Fanuc TP program (LS listing): FM113226.ls

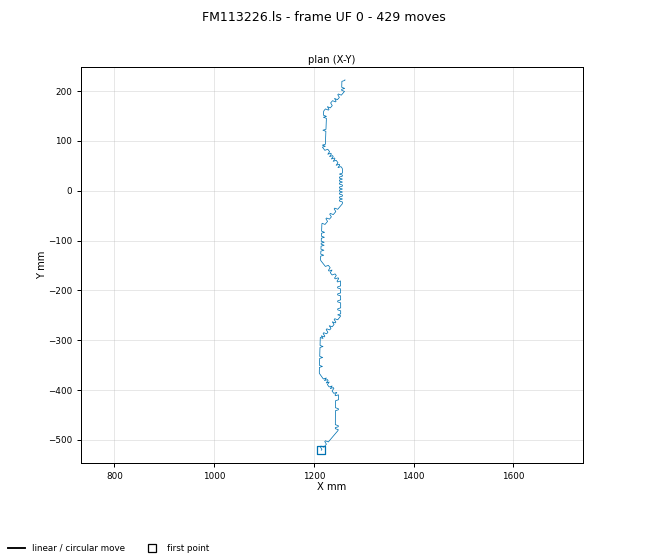
[picture p0: tool path of FM113226.ls in frame UF 0, 429 of 429 moves have a stored position in this frame; points joined in program order, loops and branches not executed]
/PROG  FM113226
/ATTR
OWNER		= MNEDITOR;
COMMENT		= "Auto FANUC move";
PROG_SIZE	= 0;
CREATE		= DATE 26-05-06  TIME 11:32:26;
MODIFIED	= DATE 26-05-06  TIME 11:32:26;
FILE_NAME	= ;
VERSION		= 0;
LINE_COUNT	= 434;
MEMORY_SIZE	= 0;
PROTECT		= READ_WRITE;
TCD:  STACK_SIZE	= 0,
      TASK_PRIORITY	= 50,
      TIME_SLICE	= 0,
      BUSY_LAMP_OFF	= 0,
      ABORT_REQUEST	= 0,
      PAUSE_REQUEST	= 0;
DEFAULT_GROUP	= 1,*,*,*,*;
CONTROL_CODE	= 00000000 00000000;
/MN
   1:  UFRAME_NUM=0 ;
   2:  UTOOL_NUM=1 ;
   3:  R[93]=10 ;
   4:  L P[1] 7mm/sec FINE ;
   5:  L P[2] 7mm/sec CNT50 ;
   6:  L P[3] 7mm/sec CNT50 ;
   7:  L P[4] 7mm/sec CNT50 ;
   8:  L P[5] 7mm/sec CNT50 ;
   9:  L P[6] 7mm/sec CNT50 ;
  10:  L P[7] 7mm/sec CNT50 ;
  11:  L P[8] 7mm/sec CNT50 ;
  12:  L P[9] 7mm/sec CNT50 ;
  13:  L P[10] 7mm/sec CNT50 ;
  14:  L P[11] 7mm/sec CNT50 ;
  15:  L P[12] 7mm/sec CNT50 ;
  16:  L P[13] 7mm/sec CNT50 ;
  17:  L P[14] 7mm/sec CNT50 ;
  18:  L P[15] 7mm/sec CNT50 ;
  19:  L P[16] 7mm/sec CNT50 ;
  20:  L P[17] 7mm/sec CNT50 ;
  21:  L P[18] 7mm/sec CNT50 ;
  22:  L P[19] 7mm/sec CNT50 ;
  23:  L P[20] 7mm/sec CNT50 ;
  24:  L P[21] 7mm/sec CNT50 ;
  25:  L P[22] 7mm/sec CNT50 ;
  26:  L P[23] 7mm/sec CNT50 ;
  27:  L P[24] 7mm/sec CNT50 ;
  28:  L P[25] 7mm/sec CNT50 ;
  29:  L P[26] 7mm/sec CNT50 ;
  30:  L P[27] 7mm/sec CNT50 ;
  31:  L P[28] 7mm/sec CNT50 ;
  32:  L P[29] 7mm/sec CNT50 ;
  33:  L P[30] 7mm/sec CNT50 ;
  34:  L P[31] 7mm/sec CNT50 ;
  35:  L P[32] 7mm/sec CNT50 ;
  36:  L P[33] 7mm/sec CNT50 ;
  37:  L P[34] 7mm/sec CNT50 ;
  38:  L P[35] 7mm/sec CNT50 ;
  39:  L P[36] 7mm/sec CNT50 ;
  40:  L P[37] 7mm/sec CNT50 ;
  41:  L P[38] 7mm/sec CNT50 ;
  42:  L P[39] 7mm/sec CNT50 ;
  43:  L P[40] 7mm/sec CNT50 ;
  44:  L P[41] 7mm/sec CNT50 ;
  45:  L P[42] 7mm/sec CNT50 ;
  46:  L P[43] 7mm/sec CNT50 ;
  47:  L P[44] 7mm/sec CNT50 ;
  48:  L P[45] 7mm/sec CNT50 ;
  49:  L P[46] 7mm/sec CNT50 ;
  50:  L P[47] 7mm/sec CNT50 ;
  51:  L P[48] 7mm/sec CNT50 ;
  52:  L P[49] 7mm/sec CNT50 ;
  53:  L P[50] 7mm/sec CNT50 ;
  54:  L P[51] 7mm/sec CNT50 ;
  55:  L P[52] 7mm/sec CNT50 ;
  56:  L P[53] 7mm/sec CNT50 ;
  57:  L P[54] 7mm/sec CNT50 ;
  58:  L P[55] 7mm/sec CNT50 ;
  59:  L P[56] 7mm/sec CNT50 ;
  60:  L P[57] 7mm/sec CNT50 ;
  61:  L P[58] 7mm/sec CNT50 ;
  62:  L P[59] 7mm/sec CNT50 ;
  63:  L P[60] 7mm/sec CNT50 ;
  64:  L P[61] 7mm/sec CNT50 ;
  65:  L P[62] 7mm/sec CNT50 ;
  66:  L P[63] 7mm/sec CNT50 ;
  67:  L P[64] 7mm/sec CNT50 ;
  68:  L P[65] 7mm/sec CNT50 ;
  69:  L P[66] 7mm/sec CNT50 ;
  70:  L P[67] 7mm/sec CNT50 ;
  71:  L P[68] 7mm/sec CNT50 ;
  72:  L P[69] 7mm/sec CNT50 ;
  73:  L P[70] 7mm/sec CNT50 ;
  74:  L P[71] 7mm/sec CNT50 ;
  75:  L P[72] 7mm/sec CNT50 ;
  76:  L P[73] 7mm/sec CNT50 ;
  77:  L P[74] 7mm/sec CNT50 ;
  78:  L P[75] 7mm/sec CNT50 ;
  79:  L P[76] 7mm/sec CNT50 ;
  80:  L P[77] 7mm/sec CNT50 ;
  81:  L P[78] 7mm/sec CNT50 ;
  82:  L P[79] 7mm/sec CNT50 ;
  83:  L P[80] 7mm/sec CNT50 ;
  84:  L P[81] 7mm/sec CNT50 ;
  85:  L P[82] 7mm/sec CNT50 ;
  86:  L P[83] 7mm/sec CNT50 ;
  87:  L P[84] 7mm/sec CNT50 ;
  88:  L P[85] 7mm/sec CNT50 ;
  89:  L P[86] 7mm/sec CNT50 ;
  90:  L P[87] 7mm/sec CNT50 ;
  91:  L P[88] 7mm/sec CNT50 ;
  92:  L P[89] 7mm/sec CNT50 ;
  93:  L P[90] 7mm/sec CNT50 ;
  94:  L P[91] 7mm/sec CNT50 ;
  95:  L P[92] 7mm/sec CNT50 ;
  96:  L P[93] 7mm/sec CNT50 ;
  97:  L P[94] 7mm/sec CNT50 ;
  98:  L P[95] 7mm/sec CNT50 ;
  99:  L P[96] 7mm/sec CNT50 ;
 100:  L P[97] 7mm/sec CNT50 ;
 101:  L P[98] 7mm/sec CNT50 ;
 102:  L P[99] 7mm/sec CNT50 ;
 103:  L P[100] 7mm/sec CNT50 ;
 104:  L P[101] 7mm/sec CNT50 ;
 105:  L P[102] 7mm/sec CNT50 ;
 106:  L P[103] 7mm/sec CNT50 ;
 107:  L P[104] 7mm/sec CNT50 ;
 108:  L P[105] 7mm/sec CNT50 ;
 109:  L P[106] 7mm/sec CNT50 ;
 110:  L P[107] 7mm/sec CNT50 ;
 111:  L P[108] 7mm/sec CNT50 ;
 112:  L P[109] 7mm/sec CNT50 ;
 113:  L P[110] 7mm/sec CNT50 ;
 114:  L P[111] 7mm/sec CNT50 ;
 115:  L P[112] 7mm/sec CNT50 ;
 116:  L P[113] 7mm/sec CNT50 ;
 117:  L P[114] 7mm/sec CNT50 ;
 118:  L P[115] 7mm/sec CNT50 ;
 119:  L P[116] 7mm/sec CNT50 ;
 120:  L P[117] 7mm/sec CNT50 ;
 121:  L P[118] 7mm/sec CNT50 ;
 122:  L P[119] 7mm/sec CNT50 ;
 123:  L P[120] 7mm/sec CNT50 ;
 124:  L P[121] 7mm/sec CNT50 ;
 125:  L P[122] 7mm/sec CNT50 ;
 126:  L P[123] 7mm/sec CNT50 ;
 127:  L P[124] 7mm/sec CNT50 ;
 128:  L P[125] 7mm/sec CNT50 ;
 129:  L P[126] 7mm/sec CNT50 ;
 130:  L P[127] 7mm/sec CNT50 ;
 131:  L P[128] 7mm/sec CNT50 ;
 132:  L P[129] 7mm/sec CNT50 ;
 133:  L P[130] 7mm/sec CNT50 ;
 134:  L P[131] 7mm/sec CNT50 ;
 135:  L P[132] 7mm/sec CNT50 ;
 136:  L P[133] 7mm/sec CNT50 ;
 137:  L P[134] 7mm/sec CNT50 ;
 138:  L P[135] 7mm/sec CNT50 ;
 139:  L P[136] 7mm/sec CNT50 ;
 140:  L P[137] 7mm/sec CNT50 ;
 141:  L P[138] 7mm/sec CNT50 ;
 142:  L P[139] 7mm/sec CNT50 ;
 143:  L P[140] 7mm/sec CNT50 ;
 144:  L P[141] 7mm/sec CNT50 ;
 145:  L P[142] 7mm/sec CNT50 ;
 146:  L P[143] 7mm/sec CNT50 ;
 147:  L P[144] 7mm/sec CNT50 ;
 148:  L P[145] 7mm/sec CNT50 ;
 149:  L P[146] 7mm/sec CNT50 ;
 150:  L P[147] 7mm/sec CNT50 ;
 151:  L P[148] 7mm/sec CNT50 ;
 152:  L P[149] 7mm/sec CNT50 ;
 153:  L P[150] 7mm/sec CNT50 ;
 154:  L P[151] 7mm/sec CNT50 ;
 155:  L P[152] 7mm/sec CNT50 ;
 156:  L P[153] 7mm/sec CNT50 ;
 157:  L P[154] 7mm/sec CNT50 ;
 158:  L P[155] 7mm/sec CNT50 ;
 159:  L P[156] 7mm/sec CNT50 ;
 160:  L P[157] 7mm/sec CNT50 ;
 161:  L P[158] 7mm/sec CNT50 ;
 162:  L P[159] 7mm/sec CNT50 ;
 163:  L P[160] 7mm/sec CNT50 ;
 164:  L P[161] 7mm/sec CNT50 ;
 165:  L P[162] 7mm/sec CNT50 ;
 166:  L P[163] 7mm/sec CNT50 ;
 167:  L P[164] 7mm/sec CNT50 ;
 168:  L P[165] 7mm/sec CNT50 ;
 169:  L P[166] 7mm/sec CNT50 ;
 170:  L P[167] 7mm/sec CNT50 ;
 171:  L P[168] 7mm/sec CNT50 ;
 172:  L P[169] 7mm/sec CNT50 ;
 173:  L P[170] 7mm/sec CNT50 ;
 174:  L P[171] 7mm/sec CNT50 ;
 175:  L P[172] 7mm/sec CNT50 ;
 176:  L P[173] 7mm/sec CNT50 ;
 177:  L P[174] 7mm/sec CNT50 ;
 178:  L P[175] 7mm/sec CNT50 ;
 179:  L P[176] 7mm/sec CNT50 ;
 180:  L P[177] 7mm/sec CNT50 ;
 181:  L P[178] 7mm/sec CNT50 ;
 182:  L P[179] 7mm/sec CNT50 ;
 183:  L P[180] 7mm/sec CNT50 ;
 184:  L P[181] 7mm/sec CNT50 ;
 185:  L P[182] 7mm/sec CNT50 ;
 186:  L P[183] 7mm/sec CNT50 ;
 187:  L P[184] 7mm/sec CNT50 ;
 188:  L P[185] 7mm/sec CNT50 ;
 189:  L P[186] 7mm/sec CNT50 ;
 190:  L P[187] 7mm/sec CNT50 ;
 191:  L P[188] 7mm/sec CNT50 ;
 192:  L P[189] 7mm/sec CNT50 ;
 193:  L P[190] 7mm/sec CNT50 ;
 194:  L P[191] 7mm/sec CNT50 ;
 195:  L P[192] 7mm/sec CNT50 ;
 196:  L P[193] 7mm/sec CNT50 ;
 197:  L P[194] 7mm/sec CNT50 ;
 198:  L P[195] 7mm/sec CNT50 ;
 199:  L P[196] 7mm/sec CNT50 ;
 200:  L P[197] 7mm/sec CNT50 ;
 201:  L P[198] 7mm/sec CNT50 ;
 202:  L P[199] 7mm/sec CNT50 ;
 203:  L P[200] 7mm/sec CNT50 ;
 204:  L P[201] 7mm/sec CNT50 ;
 205:  L P[202] 7mm/sec CNT50 ;
 206:  L P[203] 7mm/sec CNT50 ;
 207:  L P[204] 7mm/sec CNT50 ;
 208:  L P[205] 7mm/sec CNT50 ;
 209:  L P[206] 7mm/sec CNT50 ;
 210:  L P[207] 7mm/sec CNT50 ;
 211:  L P[208] 7mm/sec CNT50 ;
 212:  L P[209] 7mm/sec CNT50 ;
 213:  L P[210] 7mm/sec CNT50 ;
 214:  L P[211] 7mm/sec CNT50 ;
 215:  L P[212] 7mm/sec CNT50 ;
 216:  L P[213] 7mm/sec CNT50 ;
 217:  L P[214] 7mm/sec CNT50 ;
 218:  L P[215] 7mm/sec CNT50 ;
 219:  L P[216] 7mm/sec CNT50 ;
 220:  L P[217] 7mm/sec CNT50 ;
 221:  L P[218] 7mm/sec CNT50 ;
 222:  L P[219] 7mm/sec CNT50 ;
 223:  L P[220] 7mm/sec CNT50 ;
 224:  L P[221] 7mm/sec CNT50 ;
 225:  L P[222] 7mm/sec CNT50 ;
 226:  L P[223] 7mm/sec CNT50 ;
 227:  L P[224] 7mm/sec CNT50 ;
 228:  L P[225] 7mm/sec CNT50 ;
 229:  L P[226] 7mm/sec CNT50 ;
 230:  L P[227] 7mm/sec CNT50 ;
 231:  L P[228] 7mm/sec CNT50 ;
 232:  L P[229] 7mm/sec CNT50 ;
 233:  L P[230] 7mm/sec CNT50 ;
 234:  L P[231] 7mm/sec CNT50 ;
 235:  L P[232] 7mm/sec CNT50 ;
 236:  L P[233] 7mm/sec CNT50 ;
 237:  L P[234] 7mm/sec CNT50 ;
 238:  L P[235] 7mm/sec CNT50 ;
 239:  L P[236] 7mm/sec CNT50 ;
 240:  L P[237] 7mm/sec CNT50 ;
 241:  L P[238] 7mm/sec CNT50 ;
 242:  L P[239] 7mm/sec CNT50 ;
 243:  L P[240] 7mm/sec CNT50 ;
 244:  L P[241] 7mm/sec CNT50 ;
 245:  L P[242] 7mm/sec CNT50 ;
 246:  L P[243] 7mm/sec CNT50 ;
 247:  L P[244] 7mm/sec CNT50 ;
 248:  L P[245] 7mm/sec CNT50 ;
 249:  L P[246] 7mm/sec CNT50 ;
 250:  L P[247] 7mm/sec CNT50 ;
 251:  L P[248] 7mm/sec CNT50 ;
 252:  L P[249] 7mm/sec CNT50 ;
 253:  L P[250] 7mm/sec CNT50 ;
 254:  L P[251] 7mm/sec CNT50 ;
 255:  L P[252] 7mm/sec CNT50 ;
 256:  L P[253] 7mm/sec CNT50 ;
 257:  L P[254] 7mm/sec CNT50 ;
 258:  L P[255] 7mm/sec CNT50 ;
 259:  L P[256] 7mm/sec CNT50 ;
 260:  L P[257] 7mm/sec CNT50 ;
 261:  L P[258] 7mm/sec CNT50 ;
 262:  L P[259] 7mm/sec CNT50 ;
 263:  L P[260] 7mm/sec CNT50 ;
 264:  L P[261] 7mm/sec CNT50 ;
 265:  L P[262] 7mm/sec CNT50 ;
 266:  L P[263] 7mm/sec CNT50 ;
 267:  L P[264] 7mm/sec CNT50 ;
 268:  L P[265] 7mm/sec CNT50 ;
 269:  L P[266] 7mm/sec CNT50 ;
 270:  L P[267] 7mm/sec CNT50 ;
 271:  L P[268] 7mm/sec CNT50 ;
 272:  L P[269] 7mm/sec CNT50 ;
 273:  L P[270] 7mm/sec CNT50 ;
 274:  L P[271] 7mm/sec CNT50 ;
 275:  L P[272] 7mm/sec CNT50 ;
 276:  L P[273] 7mm/sec CNT50 ;
 277:  L P[274] 7mm/sec CNT50 ;
 278:  L P[275] 7mm/sec CNT50 ;
 279:  L P[276] 7mm/sec CNT50 ;
 280:  L P[277] 7mm/sec CNT50 ;
 281:  L P[278] 7mm/sec CNT50 ;
 282:  L P[279] 7mm/sec CNT50 ;
 283:  L P[280] 7mm/sec CNT50 ;
 284:  L P[281] 7mm/sec CNT50 ;
 285:  L P[282] 7mm/sec CNT50 ;
 286:  L P[283] 7mm/sec CNT50 ;
 287:  L P[284] 7mm/sec CNT50 ;
 288:  L P[285] 7mm/sec CNT50 ;
 289:  L P[286] 7mm/sec CNT50 ;
 290:  L P[287] 7mm/sec CNT50 ;
 291:  L P[288] 7mm/sec CNT50 ;
 292:  L P[289] 7mm/sec CNT50 ;
 293:  L P[290] 7mm/sec CNT50 ;
 294:  L P[291] 7mm/sec CNT50 ;
 295:  L P[292] 7mm/sec CNT50 ;
 296:  L P[293] 7mm/sec CNT50 ;
 297:  L P[294] 7mm/sec CNT50 ;
 298:  L P[295] 7mm/sec CNT50 ;
 299:  L P[296] 7mm/sec CNT50 ;
 300:  L P[297] 7mm/sec CNT50 ;
 301:  L P[298] 7mm/sec CNT50 ;
 302:  L P[299] 7mm/sec CNT50 ;
 303:  L P[300] 7mm/sec CNT50 ;
 304:  L P[301] 7mm/sec CNT50 ;
 305:  L P[302] 7mm/sec CNT50 ;
 306:  L P[303] 7mm/sec CNT50 ;
 307:  L P[304] 7mm/sec CNT50 ;
 308:  L P[305] 7mm/sec CNT50 ;
 309:  L P[306] 7mm/sec CNT50 ;
 310:  L P[307] 7mm/sec CNT50 ;
 311:  L P[308] 7mm/sec CNT50 ;
 312:  L P[309] 7mm/sec CNT50 ;
 313:  L P[310] 7mm/sec CNT50 ;
 314:  L P[311] 7mm/sec CNT50 ;
 315:  L P[312] 7mm/sec CNT50 ;
 316:  L P[313] 7mm/sec CNT50 ;
 317:  L P[314] 7mm/sec CNT50 ;
 318:  L P[315] 7mm/sec CNT50 ;
 319:  L P[316] 7mm/sec CNT50 ;
 320:  L P[317] 7mm/sec CNT50 ;
 321:  L P[318] 7mm/sec CNT50 ;
 322:  L P[319] 7mm/sec CNT50 ;
 323:  L P[320] 7mm/sec CNT50 ;
 324:  L P[321] 7mm/sec CNT50 ;
 325:  L P[322] 7mm/sec CNT50 ;
 326:  L P[323] 7mm/sec CNT50 ;
 327:  L P[324] 7mm/sec CNT50 ;
 328:  L P[325] 7mm/sec CNT50 ;
 329:  L P[326] 7mm/sec CNT50 ;
 330:  L P[327] 7mm/sec CNT50 ;
 331:  L P[328] 7mm/sec CNT50 ;
 332:  L P[329] 7mm/sec CNT50 ;
 333:  L P[330] 7mm/sec CNT50 ;
 334:  L P[331] 7mm/sec CNT50 ;
 335:  L P[332] 7mm/sec CNT50 ;
 336:  L P[333] 7mm/sec CNT50 ;
 337:  L P[334] 7mm/sec CNT50 ;
 338:  L P[335] 7mm/sec CNT50 ;
 339:  L P[336] 7mm/sec CNT50 ;
 340:  L P[337] 7mm/sec CNT50 ;
 341:  L P[338] 7mm/sec CNT50 ;
 342:  L P[339] 7mm/sec CNT50 ;
 343:  L P[340] 7mm/sec CNT50 ;
 344:  L P[341] 7mm/sec CNT50 ;
 345:  L P[342] 7mm/sec CNT50 ;
 346:  L P[343] 7mm/sec CNT50 ;
 347:  L P[344] 7mm/sec CNT50 ;
 348:  L P[345] 7mm/sec CNT50 ;
 349:  L P[346] 7mm/sec CNT50 ;
 350:  L P[347] 7mm/sec CNT50 ;
 351:  L P[348] 7mm/sec CNT50 ;
 352:  L P[349] 7mm/sec CNT50 ;
 353:  L P[350] 7mm/sec CNT50 ;
 354:  L P[351] 7mm/sec CNT50 ;
 355:  L P[352] 7mm/sec CNT50 ;
 356:  L P[353] 7mm/sec CNT50 ;
 357:  L P[354] 7mm/sec CNT50 ;
 358:  L P[355] 7mm/sec CNT50 ;
 359:  L P[356] 7mm/sec CNT50 ;
 360:  L P[357] 7mm/sec CNT50 ;
 361:  L P[358] 7mm/sec CNT50 ;
 362:  L P[359] 7mm/sec CNT50 ;
 363:  L P[360] 7mm/sec CNT50 ;
 364:  L P[361] 7mm/sec CNT50 ;
 365:  L P[362] 7mm/sec CNT50 ;
 366:  L P[363] 7mm/sec CNT50 ;
 367:  L P[364] 7mm/sec CNT50 ;
 368:  L P[365] 7mm/sec CNT50 ;
 369:  L P[366] 7mm/sec CNT50 ;
 370:  L P[367] 7mm/sec CNT50 ;
 371:  L P[368] 7mm/sec CNT50 ;
 372:  L P[369] 7mm/sec CNT50 ;
 373:  L P[370] 7mm/sec CNT50 ;
 374:  L P[371] 7mm/sec CNT50 ;
 375:  L P[372] 7mm/sec CNT50 ;
 376:  L P[373] 7mm/sec CNT50 ;
 377:  L P[374] 7mm/sec CNT50 ;
 378:  L P[375] 7mm/sec CNT50 ;
 379:  L P[376] 7mm/sec CNT50 ;
 380:  L P[377] 7mm/sec CNT50 ;
 381:  L P[378] 7mm/sec CNT50 ;
 382:  L P[379] 7mm/sec CNT50 ;
 383:  L P[380] 7mm/sec CNT50 ;
 384:  L P[381] 7mm/sec CNT50 ;
 385:  L P[382] 7mm/sec CNT50 ;
 386:  L P[383] 7mm/sec CNT50 ;
 387:  L P[384] 7mm/sec CNT50 ;
 388:  L P[385] 7mm/sec CNT50 ;
 389:  L P[386] 7mm/sec CNT50 ;
 390:  L P[387] 7mm/sec CNT50 ;
 391:  L P[388] 7mm/sec CNT50 ;
 392:  L P[389] 7mm/sec CNT50 ;
 393:  L P[390] 7mm/sec CNT50 ;
 394:  L P[391] 7mm/sec CNT50 ;
 395:  L P[392] 7mm/sec CNT50 ;
 396:  L P[393] 7mm/sec CNT50 ;
 397:  L P[394] 7mm/sec CNT50 ;
 398:  L P[395] 7mm/sec CNT50 ;
 399:  L P[396] 7mm/sec CNT50 ;
 400:  L P[397] 7mm/sec CNT50 ;
 401:  L P[398] 7mm/sec CNT50 ;
 402:  L P[399] 7mm/sec CNT50 ;
 403:  L P[400] 7mm/sec CNT50 ;
 404:  L P[401] 7mm/sec CNT50 ;
 405:  L P[402] 7mm/sec CNT50 ;
 406:  L P[403] 7mm/sec CNT50 ;
 407:  L P[404] 7mm/sec CNT50 ;
 408:  L P[405] 7mm/sec CNT50 ;
 409:  L P[406] 7mm/sec CNT50 ;
 410:  L P[407] 7mm/sec CNT50 ;
 411:  L P[408] 7mm/sec CNT50 ;
 412:  L P[409] 7mm/sec CNT50 ;
 413:  L P[410] 7mm/sec CNT50 ;
 414:  L P[411] 7mm/sec CNT50 ;
 415:  L P[412] 7mm/sec CNT50 ;
 416:  L P[413] 7mm/sec CNT50 ;
 417:  L P[414] 7mm/sec CNT50 ;
 418:  L P[415] 7mm/sec CNT50 ;
 419:  L P[416] 7mm/sec CNT50 ;
 420:  L P[417] 7mm/sec CNT50 ;
 421:  L P[418] 7mm/sec CNT50 ;
 422:  L P[419] 7mm/sec CNT50 ;
 423:  L P[420] 7mm/sec CNT50 ;
 424:  L P[421] 7mm/sec CNT50 ;
 425:  L P[422] 7mm/sec CNT50 ;
 426:  L P[423] 7mm/sec CNT50 ;
 427:  L P[424] 7mm/sec CNT50 ;
 428:  L P[425] 7mm/sec CNT50 ;
 429:  L P[426] 7mm/sec CNT50 ;
 430:  L P[427] 7mm/sec CNT50 ;
 431:  L P[428] 7mm/sec CNT50 ;
 432:  L P[429] 7mm/sec FINE ;
 433:  R[93]=1 ;
 434:  END ;
/POS
P[1]{
   GP1:
	UF : 0, UT : 1,		CONFIG : 'N U T, 0, 0, 0',
	X = 1214.854  mm,	Y = -520.674  mm,	Z = -244.012  mm,
	W = 0.000 deg,	P = 30.000 deg,	R = 139.708 deg
};
P[2]{
   GP1:
	UF : 0, UT : 1,		CONFIG : 'N U T, 0, 0, 0',
	X = 1216.138  mm,	Y = -519.161  mm,	Z = -244.261  mm,
	W = 0.000 deg,	P = 30.000 deg,	R = 139.708 deg
};
P[3]{
   GP1:
	UF : 0, UT : 1,		CONFIG : 'N U T, 0, 0, 0',
	X = 1212.844  mm,	Y = -513.767  mm,	Z = -244.510  mm,
	W = 0.000 deg,	P = 30.000 deg,	R = 139.708 deg
};
P[4]{
   GP1:
	UF : 0, UT : 1,		CONFIG : 'N U T, 0, 0, 0',
	X = 1214.128  mm,	Y = -512.253  mm,	Z = -244.760  mm,
	W = 0.000 deg,	P = 30.000 deg,	R = 139.708 deg
};
P[5]{
   GP1:
	UF : 0, UT : 1,		CONFIG : 'N U T, 0, 0, 0',
	X = 1219.987  mm,	Y = -514.620  mm,	Z = -245.009  mm,
	W = 0.000 deg,	P = 30.000 deg,	R = 139.708 deg
};
P[6]{
   GP1:
	UF : 0, UT : 1,		CONFIG : 'N U T, 0, 0, 0',
	X = 1221.271  mm,	Y = -513.106  mm,	Z = -245.258  mm,
	W = 0.000 deg,	P = 30.000 deg,	R = 139.708 deg
};
P[7]{
   GP1:
	UF : 0, UT : 1,		CONFIG : 'N U T, 0, 0, 0',
	X = 1222.554  mm,	Y = -511.593  mm,	Z = -245.507  mm,
	W = 0.000 deg,	P = 30.000 deg,	R = 139.708 deg
};
P[8]{
   GP1:
	UF : 0, UT : 1,		CONFIG : 'N U T, 0, 0, 0',
	X = 1223.837  mm,	Y = -510.079  mm,	Z = -245.756  mm,
	W = 0.000 deg,	P = 30.000 deg,	R = 139.708 deg
};
P[9]{
   GP1:
	UF : 0, UT : 1,		CONFIG : 'N U T, 0, 0, 0',
	X = 1225.121  mm,	Y = -508.565  mm,	Z = -246.005  mm,
	W = 0.000 deg,	P = 30.000 deg,	R = 139.708 deg
};
P[10]{
   GP1:
	UF : 0, UT : 1,		CONFIG : 'N U T, 0, 0, 0',
	X = 1221.827  mm,	Y = -503.171  mm,	Z = -246.254  mm,
	W = 0.000 deg,	P = 30.000 deg,	R = 139.708 deg
};
P[11]{
   GP1:
	UF : 0, UT : 1,		CONFIG : 'N U T, 0, 0, 0',
	X = 1223.111  mm,	Y = -501.658  mm,	Z = -246.503  mm,
	W = 0.000 deg,	P = 30.000 deg,	R = 139.708 deg
};
P[12]{
   GP1:
	UF : 0, UT : 1,		CONFIG : 'N U T, 0, 0, 0',
	X = 1228.970  mm,	Y = -504.024  mm,	Z = -246.752  mm,
	W = 0.000 deg,	P = 30.000 deg,	R = 139.708 deg
};
P[13]{
   GP1:
	UF : 0, UT : 1,		CONFIG : 'N U T, 0, 0, 0',
	X = 1230.254  mm,	Y = -502.511  mm,	Z = -247.001  mm,
	W = 0.000 deg,	P = 30.000 deg,	R = 139.708 deg
};
P[14]{
   GP1:
	UF : 0, UT : 1,		CONFIG : 'N U T, 0, 0, 0',
	X = 1231.537  mm,	Y = -500.997  mm,	Z = -247.250  mm,
	W = 0.000 deg,	P = 30.000 deg,	R = 139.708 deg
};
P[15]{
   GP1:
	UF : 0, UT : 1,		CONFIG : 'N U T, 0, 0, 0',
	X = 1232.820  mm,	Y = -499.483  mm,	Z = -247.499  mm,
	W = 0.000 deg,	P = 30.000 deg,	R = 139.708 deg
};
P[16]{
   GP1:
	UF : 0, UT : 1,		CONFIG : 'N U T, 0, 0, 0',
	X = 1234.104  mm,	Y = -497.970  mm,	Z = -247.748  mm,
	W = 0.000 deg,	P = 30.000 deg,	R = 139.708 deg
};
P[17]{
   GP1:
	UF : 0, UT : 1,		CONFIG : 'N U T, 0, 0, 0',
	X = 1235.387  mm,	Y = -496.456  mm,	Z = -247.997  mm,
	W = 0.000 deg,	P = 30.000 deg,	R = 139.708 deg
};
P[18]{
   GP1:
	UF : 0, UT : 1,		CONFIG : 'N U T, 0, 0, 0',
	X = 1236.670  mm,	Y = -494.942  mm,	Z = -248.246  mm,
	W = 0.000 deg,	P = 30.000 deg,	R = 139.708 deg
};
P[19]{
   GP1:
	UF : 0, UT : 1,		CONFIG : 'N U T, 0, 0, 0',
	X = 1237.954  mm,	Y = -493.429  mm,	Z = -248.495  mm,
	W = 0.000 deg,	P = 30.000 deg,	R = 139.708 deg
};
P[20]{
   GP1:
	UF : 0, UT : 1,		CONFIG : 'N U T, 0, 0, 0',
	X = 1239.237  mm,	Y = -491.915  mm,	Z = -248.744  mm,
	W = 0.000 deg,	P = 30.000 deg,	R = 139.708 deg
};
P[21]{
   GP1:
	UF : 0, UT : 1,		CONFIG : 'N U T, 0, 0, 0',
	X = 1240.520  mm,	Y = -490.401  mm,	Z = -248.993  mm,
	W = 0.000 deg,	P = 30.000 deg,	R = 139.708 deg
};
P[22]{
   GP1:
	UF : 0, UT : 1,		CONFIG : 'N U T, 0, 0, 0',
	X = 1241.803  mm,	Y = -488.888  mm,	Z = -249.242  mm,
	W = 0.000 deg,	P = 30.000 deg,	R = 139.708 deg
};
P[23]{
   GP1:
	UF : 0, UT : 1,		CONFIG : 'N U T, 0, 0, 0',
	X = 1243.087  mm,	Y = -487.374  mm,	Z = -249.492  mm,
	W = 0.000 deg,	P = 30.000 deg,	R = 147.699 deg
};
P[24]{
   GP1:
	UF : 0, UT : 1,		CONFIG : 'N U T, 0, 0, 0',
	X = 1244.370  mm,	Y = -485.861  mm,	Z = -249.741  mm,
	W = 0.000 deg,	P = 30.000 deg,	R = 155.690 deg
};
P[25]{
   GP1:
	UF : 0, UT : 1,		CONFIG : 'N U T, 0, 0, 0',
	X = 1245.653  mm,	Y = -484.347  mm,	Z = -249.990  mm,
	W = 0.000 deg,	P = 30.000 deg,	R = 163.681 deg
};
P[26]{
   GP1:
	UF : 0, UT : 1,		CONFIG : 'N U T, 0, 0, 0',
	X = 1246.937  mm,	Y = -482.833  mm,	Z = -250.239  mm,
	W = 0.000 deg,	P = 30.000 deg,	R = 171.672 deg
};
P[27]{
   GP1:
	UF : 0, UT : 1,		CONFIG : 'N U T, 0, 0, 0',
	X = 1248.220  mm,	Y = -481.320  mm,	Z = -250.488  mm,
	W = 0.000 deg,	P = 30.000 deg,	R = 179.663 deg
};
P[28]{
   GP1:
	UF : 0, UT : 1,		CONFIG : 'N U T, 0, 0, 0',
	X = 1248.981  mm,	Y = -479.414  mm,	Z = -250.498  mm,
	W = 0.000 deg,	P = 30.000 deg,	R = 179.663 deg
};
P[29]{
   GP1:
	UF : 0, UT : 1,		CONFIG : 'N U T, 0, 0, 0',
	X = 1242.994  mm,	Y = -477.381  mm,	Z = -250.475  mm,
	W = 0.000 deg,	P = 30.000 deg,	R = 179.663 deg
};
P[30]{
   GP1:
	UF : 0, UT : 1,		CONFIG : 'N U T, 0, 0, 0',
	X = 1243.005  mm,	Y = -475.381  mm,	Z = -250.452  mm,
	W = 0.000 deg,	P = 30.000 deg,	R = 179.663 deg
};
P[31]{
   GP1:
	UF : 0, UT : 1,		CONFIG : 'N U T, 0, 0, 0',
	X = 1249.017  mm,	Y = -473.417  mm,	Z = -250.429  mm,
	W = 0.000 deg,	P = 30.000 deg,	R = 179.663 deg
};
P[32]{
   GP1:
	UF : 0, UT : 1,		CONFIG : 'N U T, 0, 0, 0',
	X = 1249.029  mm,	Y = -471.417  mm,	Z = -250.405  mm,
	W = 0.000 deg,	P = 30.000 deg,	R = 179.663 deg
};
P[33]{
   GP1:
	UF : 0, UT : 1,		CONFIG : 'N U T, 0, 0, 0',
	X = 1243.041  mm,	Y = -469.382  mm,	Z = -250.382  mm,
	W = 0.000 deg,	P = 30.000 deg,	R = 179.663 deg
};
P[34]{
   GP1:
	UF : 0, UT : 1,		CONFIG : 'N U T, 0, 0, 0',
	X = 1243.052  mm,	Y = -467.382  mm,	Z = -250.359  mm,
	W = 0.000 deg,	P = 30.000 deg,	R = 179.663 deg
};
P[35]{
   GP1:
	UF : 0, UT : 1,		CONFIG : 'N U T, 0, 0, 0',
	X = 1243.064  mm,	Y = -465.382  mm,	Z = -250.336  mm,
	W = 0.000 deg,	P = 30.000 deg,	R = 179.663 deg
};
P[36]{
   GP1:
	UF : 0, UT : 1,		CONFIG : 'N U T, 0, 0, 0',
	X = 1243.076  mm,	Y = -463.382  mm,	Z = -250.312  mm,
	W = 0.000 deg,	P = 30.000 deg,	R = 179.663 deg
};
P[37]{
   GP1:
	UF : 0, UT : 1,		CONFIG : 'N U T, 0, 0, 0',
	X = 1243.088  mm,	Y = -461.383  mm,	Z = -250.289  mm,
	W = 0.000 deg,	P = 30.000 deg,	R = 179.663 deg
};
P[38]{
   GP1:
	UF : 0, UT : 1,		CONFIG : 'N U T, 0, 0, 0',
	X = 1243.100  mm,	Y = -459.383  mm,	Z = -250.266  mm,
	W = 0.000 deg,	P = 30.000 deg,	R = 179.663 deg
};
P[39]{
   GP1:
	UF : 0, UT : 1,		CONFIG : 'N U T, 0, 0, 0',
	X = 1243.111  mm,	Y = -457.383  mm,	Z = -250.243  mm,
	W = 0.000 deg,	P = 30.000 deg,	R = 179.663 deg
};
P[40]{
   GP1:
	UF : 0, UT : 1,		CONFIG : 'N U T, 0, 0, 0',
	X = 1243.123  mm,	Y = -455.383  mm,	Z = -250.219  mm,
	W = 0.000 deg,	P = 30.000 deg,	R = 179.663 deg
};
P[41]{
   GP1:
	UF : 0, UT : 1,		CONFIG : 'N U T, 0, 0, 0',
	X = 1243.135  mm,	Y = -453.383  mm,	Z = -250.196  mm,
	W = 0.000 deg,	P = 30.000 deg,	R = 179.663 deg
};
P[42]{
   GP1:
	UF : 0, UT : 1,		CONFIG : 'N U T, 0, 0, 0',
	X = 1243.147  mm,	Y = -451.383  mm,	Z = -250.173  mm,
	W = 0.000 deg,	P = 30.000 deg,	R = 179.663 deg
};
P[43]{
   GP1:
	UF : 0, UT : 1,		CONFIG : 'N U T, 0, 0, 0',
	X = 1243.158  mm,	Y = -449.384  mm,	Z = -250.149  mm,
	W = 0.000 deg,	P = 30.000 deg,	R = 179.663 deg
};
P[44]{
   GP1:
	UF : 0, UT : 1,		CONFIG : 'N U T, 0, 0, 0',
	X = 1243.170  mm,	Y = -447.384  mm,	Z = -250.126  mm,
	W = 0.000 deg,	P = 30.000 deg,	R = 179.663 deg
};
P[45]{
   GP1:
	UF : 0, UT : 1,		CONFIG : 'N U T, 0, 0, 0',
	X = 1243.182  mm,	Y = -445.384  mm,	Z = -250.103  mm,
	W = 0.000 deg,	P = 30.000 deg,	R = 179.663 deg
};
P[46]{
   GP1:
	UF : 0, UT : 1,		CONFIG : 'N U T, 0, 0, 0',
	X = 1243.194  mm,	Y = -443.384  mm,	Z = -250.080  mm,
	W = 0.000 deg,	P = 30.000 deg,	R = 179.663 deg
};
P[47]{
   GP1:
	UF : 0, UT : 1,		CONFIG : 'N U T, 0, 0, 0',
	X = 1243.205  mm,	Y = -441.384  mm,	Z = -250.056  mm,
	W = 0.000 deg,	P = 30.000 deg,	R = 179.663 deg
};
P[48]{
   GP1:
	UF : 0, UT : 1,		CONFIG : 'N U T, 0, 0, 0',
	X = 1249.217  mm,	Y = -439.420  mm,	Z = -250.033  mm,
	W = 0.000 deg,	P = 30.000 deg,	R = 179.663 deg
};
P[49]{
   GP1:
	UF : 0, UT : 1,		CONFIG : 'N U T, 0, 0, 0',
	X = 1249.229  mm,	Y = -437.420  mm,	Z = -250.010  mm,
	W = 0.000 deg,	P = 30.000 deg,	R = 179.663 deg
};
P[50]{
   GP1:
	UF : 0, UT : 1,		CONFIG : 'N U T, 0, 0, 0',
	X = 1243.241  mm,	Y = -435.385  mm,	Z = -249.987  mm,
	W = 0.000 deg,	P = 30.000 deg,	R = 179.663 deg
};
P[51]{
   GP1:
	UF : 0, UT : 1,		CONFIG : 'N U T, 0, 0, 0',
	X = 1243.253  mm,	Y = -433.385  mm,	Z = -249.963  mm,
	W = 0.000 deg,	P = 30.000 deg,	R = 179.663 deg
};
P[52]{
   GP1:
	UF : 0, UT : 1,		CONFIG : 'N U T, 0, 0, 0',
	X = 1243.264  mm,	Y = -431.385  mm,	Z = -249.940  mm,
	W = 0.000 deg,	P = 30.000 deg,	R = 179.663 deg
};
P[53]{
   GP1:
	UF : 0, UT : 1,		CONFIG : 'N U T, 0, 0, 0',
	X = 1243.276  mm,	Y = -429.385  mm,	Z = -249.917  mm,
	W = 0.000 deg,	P = 30.000 deg,	R = 179.663 deg
};
P[54]{
   GP1:
	UF : 0, UT : 1,		CONFIG : 'N U T, 0, 0, 0',
	X = 1243.288  mm,	Y = -427.385  mm,	Z = -249.894  mm,
	W = 0.000 deg,	P = 30.000 deg,	R = 179.663 deg
};
P[55]{
   GP1:
	UF : 0, UT : 1,		CONFIG : 'N U T, 0, 0, 0',
	X = 1243.300  mm,	Y = -425.386  mm,	Z = -249.870  mm,
	W = 0.000 deg,	P = 30.000 deg,	R = 179.663 deg
};
P[56]{
   GP1:
	UF : 0, UT : 1,		CONFIG : 'N U T, 0, 0, 0',
	X = 1243.311  mm,	Y = -423.386  mm,	Z = -249.847  mm,
	W = 0.000 deg,	P = 30.000 deg,	R = 179.663 deg
};
P[57]{
   GP1:
	UF : 0, UT : 1,		CONFIG : 'N U T, 0, 0, 0',
	X = 1243.323  mm,	Y = -421.386  mm,	Z = -249.824  mm,
	W = 0.000 deg,	P = 30.000 deg,	R = 179.663 deg
};
P[58]{
   GP1:
	UF : 0, UT : 1,		CONFIG : 'N U T, 0, 0, 0',
	X = 1249.335  mm,	Y = -419.421  mm,	Z = -249.800  mm,
	W = 0.000 deg,	P = 30.000 deg,	R = -173.342 deg
};
P[59]{
   GP1:
	UF : 0, UT : 1,		CONFIG : 'N U T, 0, 0, 0',
	X = 1249.347  mm,	Y = -417.422  mm,	Z = -249.777  mm,
	W = 0.000 deg,	P = 30.000 deg,	R = -166.059 deg
};
P[60]{
   GP1:
	UF : 0, UT : 1,		CONFIG : 'N U T, 0, 0, 0',
	X = 1249.358  mm,	Y = -415.422  mm,	Z = -249.754  mm,
	W = 0.000 deg,	P = 30.000 deg,	R = -158.776 deg
};
P[61]{
   GP1:
	UF : 0, UT : 1,		CONFIG : 'N U T, 0, 0, 0',
	X = 1249.370  mm,	Y = -413.422  mm,	Z = -249.731  mm,
	W = 0.000 deg,	P = 30.000 deg,	R = -151.493 deg
};
P[62]{
   GP1:
	UF : 0, UT : 1,		CONFIG : 'N U T, 0, 0, 0',
	X = 1249.382  mm,	Y = -411.422  mm,	Z = -249.707  mm,
	W = 0.000 deg,	P = 30.000 deg,	R = -144.211 deg
};
P[63]{
   GP1:
	UF : 0, UT : 1,		CONFIG : 'N U T, 0, 0, 0',
	X = 1249.288  mm,	Y = -409.480  mm,	Z = -249.694  mm,
	W = 0.000 deg,	P = 30.000 deg,	R = -143.923 deg
};
P[64]{
   GP1:
	UF : 0, UT : 1,		CONFIG : 'N U T, 0, 0, 0',
	X = 1243.470  mm,	Y = -411.339  mm,	Z = -249.584  mm,
	W = 0.000 deg,	P = 30.000 deg,	R = -143.923 deg
};
P[65]{
   GP1:
	UF : 0, UT : 1,		CONFIG : 'N U T, 0, 0, 0',
	X = 1242.302  mm,	Y = -409.737  mm,	Z = -249.324  mm,
	W = 0.000 deg,	P = 30.000 deg,	R = -143.923 deg
};
P[66]{
   GP1:
	UF : 0, UT : 1,		CONFIG : 'N U T, 0, 0, 0',
	X = 1245.984  mm,	Y = -404.601  mm,	Z = -249.064  mm,
	W = 0.000 deg,	P = 30.000 deg,	R = -143.923 deg
};
P[67]{
   GP1:
	UF : 0, UT : 1,		CONFIG : 'N U T, 0, 0, 0',
	X = 1239.967  mm,	Y = -406.531  mm,	Z = -248.804  mm,
	W = 0.000 deg,	P = 30.000 deg,	R = -143.923 deg
};
P[68]{
   GP1:
	UF : 0, UT : 1,		CONFIG : 'N U T, 0, 0, 0',
	X = 1238.799  mm,	Y = -404.928  mm,	Z = -248.545  mm,
	W = 0.000 deg,	P = 30.000 deg,	R = -143.923 deg
};
P[69]{
   GP1:
	UF : 0, UT : 1,		CONFIG : 'N U T, 0, 0, 0',
	X = 1237.631  mm,	Y = -403.325  mm,	Z = -248.285  mm,
	W = 0.000 deg,	P = 30.000 deg,	R = -143.923 deg
};
P[70]{
   GP1:
	UF : 0, UT : 1,		CONFIG : 'N U T, 0, 0, 0',
	X = 1236.464  mm,	Y = -401.723  mm,	Z = -248.025  mm,
	W = 0.000 deg,	P = 30.000 deg,	R = -143.923 deg
};
P[71]{
   GP1:
	UF : 0, UT : 1,		CONFIG : 'N U T, 0, 0, 0',
	X = 1240.145  mm,	Y = -396.587  mm,	Z = -247.765  mm,
	W = 0.000 deg,	P = 30.000 deg,	R = -143.923 deg
};
P[72]{
   GP1:
	UF : 0, UT : 1,		CONFIG : 'N U T, 0, 0, 0',
	X = 1238.977  mm,	Y = -394.984  mm,	Z = -247.505  mm,
	W = 0.000 deg,	P = 30.000 deg,	R = -143.923 deg
};
P[73]{
   GP1:
	UF : 0, UT : 1,		CONFIG : 'N U T, 0, 0, 0',
	X = 1232.960  mm,	Y = -396.914  mm,	Z = -247.245  mm,
	W = 0.000 deg,	P = 30.000 deg,	R = -143.923 deg
};
P[74]{
   GP1:
	UF : 0, UT : 1,		CONFIG : 'N U T, 0, 0, 0',
	X = 1236.642  mm,	Y = -391.778  mm,	Z = -246.985  mm,
	W = 0.000 deg,	P = 30.000 deg,	R = -143.923 deg
};
P[75]{
   GP1:
	UF : 0, UT : 1,		CONFIG : 'N U T, 0, 0, 0',
	X = 1230.625  mm,	Y = -393.709  mm,	Z = -246.726  mm,
	W = 0.000 deg,	P = 30.000 deg,	R = -143.923 deg
};
P[76]{
   GP1:
	UF : 0, UT : 1,		CONFIG : 'N U T, 0, 0, 0',
	X = 1229.457  mm,	Y = -392.106  mm,	Z = -246.466  mm,
	W = 0.000 deg,	P = 30.000 deg,	R = -143.923 deg
};
P[77]{
   GP1:
	UF : 0, UT : 1,		CONFIG : 'N U T, 0, 0, 0',
	X = 1228.289  mm,	Y = -390.503  mm,	Z = -246.206  mm,
	W = 0.000 deg,	P = 30.000 deg,	R = -143.923 deg
};
P[78]{
   GP1:
	UF : 0, UT : 1,		CONFIG : 'N U T, 0, 0, 0',
	X = 1227.121  mm,	Y = -388.901  mm,	Z = -245.946  mm,
	W = 0.000 deg,	P = 30.000 deg,	R = -143.923 deg
};
P[79]{
   GP1:
	UF : 0, UT : 1,		CONFIG : 'N U T, 0, 0, 0',
	X = 1230.803  mm,	Y = -383.765  mm,	Z = -245.686  mm,
	W = 0.000 deg,	P = 30.000 deg,	R = -143.923 deg
};
P[80]{
   GP1:
	UF : 0, UT : 1,		CONFIG : 'N U T, 0, 0, 0',
	X = 1224.786  mm,	Y = -385.695  mm,	Z = -245.426  mm,
	W = 0.000 deg,	P = 30.000 deg,	R = -143.923 deg
};
P[81]{
   GP1:
	UF : 0, UT : 1,		CONFIG : 'N U T, 0, 0, 0',
	X = 1228.468  mm,	Y = -380.559  mm,	Z = -245.166  mm,
	W = 0.000 deg,	P = 30.000 deg,	R = -143.923 deg
};
P[82]{
   GP1:
	UF : 0, UT : 1,		CONFIG : 'N U T, 0, 0, 0',
	X = 1227.300  mm,	Y = -378.956  mm,	Z = -244.907  mm,
	W = 0.000 deg,	P = 30.000 deg,	R = -143.923 deg
};
P[83]{
   GP1:
	UF : 0, UT : 1,		CONFIG : 'N U T, 0, 0, 0',
	X = 1221.283  mm,	Y = -380.887  mm,	Z = -244.647  mm,
	W = 0.000 deg,	P = 30.000 deg,	R = -143.923 deg
};
P[84]{
   GP1:
	UF : 0, UT : 1,		CONFIG : 'N U T, 0, 0, 0',
	X = 1224.964  mm,	Y = -375.751  mm,	Z = -244.387  mm,
	W = 0.000 deg,	P = 30.000 deg,	R = -143.923 deg
};
P[85]{
   GP1:
	UF : 0, UT : 1,		CONFIG : 'N U T, 0, 0, 0',
	X = 1218.947  mm,	Y = -377.681  mm,	Z = -244.127  mm,
	W = 0.000 deg,	P = 30.000 deg,	R = -143.923 deg
};
P[86]{
   GP1:
	UF : 0, UT : 1,		CONFIG : 'N U T, 0, 0, 0',
	X = 1217.779  mm,	Y = -376.079  mm,	Z = -243.867  mm,
	W = 0.000 deg,	P = 30.000 deg,	R = -143.923 deg
};
P[87]{
   GP1:
	UF : 0, UT : 1,		CONFIG : 'N U T, 0, 0, 0',
	X = 1216.612  mm,	Y = -374.476  mm,	Z = -243.607  mm,
	W = 0.000 deg,	P = 30.000 deg,	R = -154.648 deg
};
P[88]{
   GP1:
	UF : 0, UT : 1,		CONFIG : 'N U T, 0, 0, 0',
	X = 1215.444  mm,	Y = -372.873  mm,	Z = -243.347  mm,
	W = 0.000 deg,	P = 30.000 deg,	R = -162.185 deg
};
P[89]{
   GP1:
	UF : 0, UT : 1,		CONFIG : 'N U T, 0, 0, 0',
	X = 1214.276  mm,	Y = -371.270  mm,	Z = -243.088  mm,
	W = 0.000 deg,	P = 30.000 deg,	R = -169.721 deg
};
P[90]{
   GP1:
	UF : 0, UT : 1,		CONFIG : 'N U T, 0, 0, 0',
	X = 1213.108  mm,	Y = -369.668  mm,	Z = -242.828  mm,
	W = 0.000 deg,	P = 30.000 deg,	R = -177.258 deg
};
P[91]{
   GP1:
	UF : 0, UT : 1,		CONFIG : 'N U T, 0, 0, 0',
	X = 1211.941  mm,	Y = -368.065  mm,	Z = -242.568  mm,
	W = 0.000 deg,	P = 30.000 deg,	R = 178.394 deg
};
P[92]{
   GP1:
	UF : 0, UT : 1,		CONFIG : 'N U T, 0, 0, 0',
	X = 1210.932  mm,	Y = -366.371  mm,	Z = -242.446  mm,
	W = 0.000 deg,	P = 30.000 deg,	R = 178.394 deg
};
P[93]{
   GP1:
	UF : 0, UT : 1,		CONFIG : 'N U T, 0, 0, 0',
	X = 1210.847  mm,	Y = -364.401  mm,	Z = -242.440  mm,
	W = 0.000 deg,	P = 30.000 deg,	R = 178.394 deg
};
P[94]{
   GP1:
	UF : 0, UT : 1,		CONFIG : 'N U T, 0, 0, 0',
	X = 1210.903  mm,	Y = -362.402  mm,	Z = -242.428  mm,
	W = 0.000 deg,	P = 30.000 deg,	R = 178.394 deg
};
P[95]{
   GP1:
	UF : 0, UT : 1,		CONFIG : 'N U T, 0, 0, 0',
	X = 1210.959  mm,	Y = -360.403  mm,	Z = -242.416  mm,
	W = 0.000 deg,	P = 30.000 deg,	R = 178.394 deg
};
P[96]{
   GP1:
	UF : 0, UT : 1,		CONFIG : 'N U T, 0, 0, 0',
	X = 1211.016  mm,	Y = -358.404  mm,	Z = -242.404  mm,
	W = 0.000 deg,	P = 30.000 deg,	R = 178.394 deg
};
P[97]{
   GP1:
	UF : 0, UT : 1,		CONFIG : 'N U T, 0, 0, 0',
	X = 1211.072  mm,	Y = -356.405  mm,	Z = -242.393  mm,
	W = 0.000 deg,	P = 30.000 deg,	R = 178.394 deg
};
P[98]{
   GP1:
	UF : 0, UT : 1,		CONFIG : 'N U T, 0, 0, 0',
	X = 1211.128  mm,	Y = -354.405  mm,	Z = -242.381  mm,
	W = 0.000 deg,	P = 30.000 deg,	R = 178.394 deg
};
P[99]{
   GP1:
	UF : 0, UT : 1,		CONFIG : 'N U T, 0, 0, 0',
	X = 1217.181  mm,	Y = -352.574  mm,	Z = -242.369  mm,
	W = 0.000 deg,	P = 30.000 deg,	R = 178.394 deg
};
P[100]{
   GP1:
	UF : 0, UT : 1,		CONFIG : 'N U T, 0, 0, 0',
	X = 1211.240  mm,	Y = -350.407  mm,	Z = -242.358  mm,
	W = 0.000 deg,	P = 30.000 deg,	R = 178.394 deg
};
P[101]{
   GP1:
	UF : 0, UT : 1,		CONFIG : 'N U T, 0, 0, 0',
	X = 1211.296  mm,	Y = -348.408  mm,	Z = -242.346  mm,
	W = 0.000 deg,	P = 30.000 deg,	R = 178.394 deg
};
P[102]{
   GP1:
	UF : 0, UT : 1,		CONFIG : 'N U T, 0, 0, 0',
	X = 1211.352  mm,	Y = -346.409  mm,	Z = -242.334  mm,
	W = 0.000 deg,	P = 30.000 deg,	R = 178.394 deg
};
P[103]{
   GP1:
	UF : 0, UT : 1,		CONFIG : 'N U T, 0, 0, 0',
	X = 1211.408  mm,	Y = -344.410  mm,	Z = -242.323  mm,
	W = 0.000 deg,	P = 30.000 deg,	R = 178.394 deg
};
P[104]{
   GP1:
	UF : 0, UT : 1,		CONFIG : 'N U T, 0, 0, 0',
	X = 1211.464  mm,	Y = -342.410  mm,	Z = -242.311  mm,
	W = 0.000 deg,	P = 30.000 deg,	R = 178.394 deg
};
P[105]{
   GP1:
	UF : 0, UT : 1,		CONFIG : 'N U T, 0, 0, 0',
	X = 1211.520  mm,	Y = -340.411  mm,	Z = -242.299  mm,
	W = 0.000 deg,	P = 30.000 deg,	R = 178.394 deg
};
P[106]{
   GP1:
	UF : 0, UT : 1,		CONFIG : 'N U T, 0, 0, 0',
	X = 1211.576  mm,	Y = -338.412  mm,	Z = -242.288  mm,
	W = 0.000 deg,	P = 30.000 deg,	R = 178.394 deg
};
P[107]{
   GP1:
	UF : 0, UT : 1,		CONFIG : 'N U T, 0, 0, 0',
	X = 1211.632  mm,	Y = -336.413  mm,	Z = -242.276  mm,
	W = 0.000 deg,	P = 30.000 deg,	R = 178.394 deg
};
P[108]{
   GP1:
	UF : 0, UT : 1,		CONFIG : 'N U T, 0, 0, 0',
	X = 1217.686  mm,	Y = -334.582  mm,	Z = -242.264  mm,
	W = 0.000 deg,	P = 30.000 deg,	R = 178.394 deg
};
P[109]{
   GP1:
	UF : 0, UT : 1,		CONFIG : 'N U T, 0, 0, 0',
	X = 1211.744  mm,	Y = -332.414  mm,	Z = -242.252  mm,
	W = 0.000 deg,	P = 30.000 deg,	R = 178.394 deg
};
P[110]{
   GP1:
	UF : 0, UT : 1,		CONFIG : 'N U T, 0, 0, 0',
	X = 1211.800  mm,	Y = -330.415  mm,	Z = -242.241  mm,
	W = 0.000 deg,	P = 30.000 deg,	R = 178.394 deg
};
P[111]{
   GP1:
	UF : 0, UT : 1,		CONFIG : 'N U T, 0, 0, 0',
	X = 1211.856  mm,	Y = -328.416  mm,	Z = -242.229  mm,
	W = 0.000 deg,	P = 30.000 deg,	R = 178.394 deg
};
P[112]{
   GP1:
	UF : 0, UT : 1,		CONFIG : 'N U T, 0, 0, 0',
	X = 1211.912  mm,	Y = -326.417  mm,	Z = -242.217  mm,
	W = 0.000 deg,	P = 30.000 deg,	R = 178.394 deg
};
P[113]{
   GP1:
	UF : 0, UT : 1,		CONFIG : 'N U T, 0, 0, 0',
	X = 1211.968  mm,	Y = -324.418  mm,	Z = -242.206  mm,
	W = 0.000 deg,	P = 30.000 deg,	R = 178.394 deg
};
P[114]{
   GP1:
	UF : 0, UT : 1,		CONFIG : 'N U T, 0, 0, 0',
	X = 1212.024  mm,	Y = -322.419  mm,	Z = -242.194  mm,
	W = 0.000 deg,	P = 30.000 deg,	R = 178.394 deg
};
P[115]{
   GP1:
	UF : 0, UT : 1,		CONFIG : 'N U T, 0, 0, 0',
	X = 1212.080  mm,	Y = -320.419  mm,	Z = -242.182  mm,
	W = 0.000 deg,	P = 30.000 deg,	R = 178.394 deg
};
P[116]{
   GP1:
	UF : 0, UT : 1,		CONFIG : 'N U T, 0, 0, 0',
	X = 1212.136  mm,	Y = -318.420  mm,	Z = -242.171  mm,
	W = 0.000 deg,	P = 30.000 deg,	R = 178.394 deg
};
P[117]{
   GP1:
	UF : 0, UT : 1,		CONFIG : 'N U T, 0, 0, 0',
	X = 1212.192  mm,	Y = -316.421  mm,	Z = -242.159  mm,
	W = 0.000 deg,	P = 30.000 deg,	R = 178.394 deg
};
P[118]{
   GP1:
	UF : 0, UT : 1,		CONFIG : 'N U T, 0, 0, 0',
	X = 1212.249  mm,	Y = -314.422  mm,	Z = -242.147  mm,
	W = 0.000 deg,	P = 30.000 deg,	R = 178.394 deg
};
P[119]{
   GP1:
	UF : 0, UT : 1,		CONFIG : 'N U T, 0, 0, 0',
	X = 1218.302  mm,	Y = -312.591  mm,	Z = -242.135  mm,
	W = 0.000 deg,	P = 30.000 deg,	R = 178.394 deg
};
P[120]{
   GP1:
	UF : 0, UT : 1,		CONFIG : 'N U T, 0, 0, 0',
	X = 1212.361  mm,	Y = -310.423  mm,	Z = -242.124  mm,
	W = 0.000 deg,	P = 30.000 deg,	R = 178.394 deg
};
P[121]{
   GP1:
	UF : 0, UT : 1,		CONFIG : 'N U T, 0, 0, 0',
	X = 1212.417  mm,	Y = -308.424  mm,	Z = -242.112  mm,
	W = 0.000 deg,	P = 30.000 deg,	R = 178.394 deg
};
P[122]{
   GP1:
	UF : 0, UT : 1,		CONFIG : 'N U T, 0, 0, 0',
	X = 1212.473  mm,	Y = -306.425  mm,	Z = -242.100  mm,
	W = 0.000 deg,	P = 30.000 deg,	R = 178.394 deg
};
P[123]{
   GP1:
	UF : 0, UT : 1,		CONFIG : 'N U T, 0, 0, 0',
	X = 1212.529  mm,	Y = -304.426  mm,	Z = -242.089  mm,
	W = 0.000 deg,	P = 30.000 deg,	R = 174.516 deg
};
P[124]{
   GP1:
	UF : 0, UT : 1,		CONFIG : 'N U T, 0, 0, 0',
	X = 1212.585  mm,	Y = -302.427  mm,	Z = -242.077  mm,
	W = 0.000 deg,	P = 30.000 deg,	R = 167.199 deg
};
P[125]{
   GP1:
	UF : 0, UT : 1,		CONFIG : 'N U T, 0, 0, 0',
	X = 1212.641  mm,	Y = -300.428  mm,	Z = -242.065  mm,
	W = 0.000 deg,	P = 30.000 deg,	R = 159.881 deg
};
P[126]{
   GP1:
	UF : 0, UT : 1,		CONFIG : 'N U T, 0, 0, 0',
	X = 1212.697  mm,	Y = -298.428  mm,	Z = -242.054  mm,
	W = 0.000 deg,	P = 30.000 deg,	R = 152.564 deg
};
P[127]{
   GP1:
	UF : 0, UT : 1,		CONFIG : 'N U T, 0, 0, 0',
	X = 1212.753  mm,	Y = -296.429  mm,	Z = -242.042  mm,
	W = 0.000 deg,	P = 30.000 deg,	R = 145.247 deg
};
P[128]{
   GP1:
	UF : 0, UT : 1,		CONFIG : 'N U T, 0, 0, 0',
	X = 1212.819  mm,	Y = -294.456  mm,	Z = -242.032  mm,
	W = 0.000 deg,	P = 30.000 deg,	R = 141.808 deg
};
P[129]{
   GP1:
	UF : 0, UT : 1,		CONFIG : 'N U T, 0, 0, 0',
	X = 1218.332  mm,	Y = -296.431  mm,	Z = -242.065  mm,
	W = 0.000 deg,	P = 30.000 deg,	R = 141.808 deg
};
P[130]{
   GP1:
	UF : 0, UT : 1,		CONFIG : 'N U T, 0, 0, 0',
	X = 1214.845  mm,	Y = -291.160  mm,	Z = -242.297  mm,
	W = 0.000 deg,	P = 30.000 deg,	R = 141.808 deg
};
P[131]{
   GP1:
	UF : 0, UT : 1,		CONFIG : 'N U T, 0, 0, 0',
	X = 1220.789  mm,	Y = -293.309  mm,	Z = -242.528  mm,
	W = 0.000 deg,	P = 30.000 deg,	R = 141.808 deg
};
P[132]{
   GP1:
	UF : 0, UT : 1,		CONFIG : 'N U T, 0, 0, 0',
	X = 1222.017  mm,	Y = -291.747  mm,	Z = -242.760  mm,
	W = 0.000 deg,	P = 30.000 deg,	R = 141.808 deg
};
P[133]{
   GP1:
	UF : 0, UT : 1,		CONFIG : 'N U T, 0, 0, 0',
	X = 1218.530  mm,	Y = -286.476  mm,	Z = -242.992  mm,
	W = 0.000 deg,	P = 30.000 deg,	R = 141.808 deg
};
P[134]{
   GP1:
	UF : 0, UT : 1,		CONFIG : 'N U T, 0, 0, 0',
	X = 1219.758  mm,	Y = -284.915  mm,	Z = -243.224  mm,
	W = 0.000 deg,	P = 30.000 deg,	R = 141.808 deg
};
P[135]{
   GP1:
	UF : 0, UT : 1,		CONFIG : 'N U T, 0, 0, 0',
	X = 1225.702  mm,	Y = -287.063  mm,	Z = -243.455  mm,
	W = 0.000 deg,	P = 30.000 deg,	R = 141.808 deg
};
P[136]{
   GP1:
	UF : 0, UT : 1,		CONFIG : 'N U T, 0, 0, 0',
	X = 1226.930  mm,	Y = -285.502  mm,	Z = -243.687  mm,
	W = 0.000 deg,	P = 30.000 deg,	R = 141.808 deg
};
P[137]{
   GP1:
	UF : 0, UT : 1,		CONFIG : 'N U T, 0, 0, 0',
	X = 1228.158  mm,	Y = -283.941  mm,	Z = -243.919  mm,
	W = 0.000 deg,	P = 30.000 deg,	R = 141.808 deg
};
P[138]{
   GP1:
	UF : 0, UT : 1,		CONFIG : 'N U T, 0, 0, 0',
	X = 1224.671  mm,	Y = -278.670  mm,	Z = -244.151  mm,
	W = 0.000 deg,	P = 30.000 deg,	R = 141.808 deg
};
P[139]{
   GP1:
	UF : 0, UT : 1,		CONFIG : 'N U T, 0, 0, 0',
	X = 1225.899  mm,	Y = -277.108  mm,	Z = -244.383  mm,
	W = 0.000 deg,	P = 30.000 deg,	R = 141.808 deg
};
P[140]{
   GP1:
	UF : 0, UT : 1,		CONFIG : 'N U T, 0, 0, 0',
	X = 1231.843  mm,	Y = -279.257  mm,	Z = -244.614  mm,
	W = 0.000 deg,	P = 30.000 deg,	R = 141.808 deg
};
P[141]{
   GP1:
	UF : 0, UT : 1,		CONFIG : 'N U T, 0, 0, 0',
	X = 1233.071  mm,	Y = -277.696  mm,	Z = -244.846  mm,
	W = 0.000 deg,	P = 30.000 deg,	R = 141.808 deg
};
P[142]{
   GP1:
	UF : 0, UT : 1,		CONFIG : 'N U T, 0, 0, 0',
	X = 1234.300  mm,	Y = -276.134  mm,	Z = -245.078  mm,
	W = 0.000 deg,	P = 30.000 deg,	R = 141.808 deg
};
P[143]{
   GP1:
	UF : 0, UT : 1,		CONFIG : 'N U T, 0, 0, 0',
	X = 1230.812  mm,	Y = -270.863  mm,	Z = -245.310  mm,
	W = 0.000 deg,	P = 30.000 deg,	R = 141.808 deg
};
P[144]{
   GP1:
	UF : 0, UT : 1,		CONFIG : 'N U T, 0, 0, 0',
	X = 1236.756  mm,	Y = -273.012  mm,	Z = -245.541  mm,
	W = 0.000 deg,	P = 30.000 deg,	R = 141.808 deg
};
P[145]{
   GP1:
	UF : 0, UT : 1,		CONFIG : 'N U T, 0, 0, 0',
	X = 1237.984  mm,	Y = -271.450  mm,	Z = -245.773  mm,
	W = 0.000 deg,	P = 30.000 deg,	R = 141.808 deg
};
P[146]{
   GP1:
	UF : 0, UT : 1,		CONFIG : 'N U T, 0, 0, 0',
	X = 1239.213  mm,	Y = -269.889  mm,	Z = -246.005  mm,
	W = 0.000 deg,	P = 30.000 deg,	R = 141.808 deg
};
P[147]{
   GP1:
	UF : 0, UT : 1,		CONFIG : 'N U T, 0, 0, 0',
	X = 1240.441  mm,	Y = -268.328  mm,	Z = -246.237  mm,
	W = 0.000 deg,	P = 30.000 deg,	R = 141.808 deg
};
P[148]{
   GP1:
	UF : 0, UT : 1,		CONFIG : 'N U T, 0, 0, 0',
	X = 1236.954  mm,	Y = -263.057  mm,	Z = -246.468  mm,
	W = 0.000 deg,	P = 30.000 deg,	R = 141.808 deg
};
P[149]{
   GP1:
	UF : 0, UT : 1,		CONFIG : 'N U T, 0, 0, 0',
	X = 1242.898  mm,	Y = -265.205  mm,	Z = -246.700  mm,
	W = 0.000 deg,	P = 30.000 deg,	R = 141.808 deg
};
P[150]{
   GP1:
	UF : 0, UT : 1,		CONFIG : 'N U T, 0, 0, 0',
	X = 1244.126  mm,	Y = -263.644  mm,	Z = -246.932  mm,
	W = 0.000 deg,	P = 30.000 deg,	R = 141.808 deg
};
P[151]{
   GP1:
	UF : 0, UT : 1,		CONFIG : 'N U T, 0, 0, 0',
	X = 1240.638  mm,	Y = -258.373  mm,	Z = -247.164  mm,
	W = 0.000 deg,	P = 30.000 deg,	R = 141.808 deg
};
P[152]{
   GP1:
	UF : 0, UT : 1,		CONFIG : 'N U T, 0, 0, 0',
	X = 1241.867  mm,	Y = -256.812  mm,	Z = -247.396  mm,
	W = 0.000 deg,	P = 30.000 deg,	R = 141.808 deg
};
P[153]{
   GP1:
	UF : 0, UT : 1,		CONFIG : 'N U T, 0, 0, 0',
	X = 1247.811  mm,	Y = -258.960  mm,	Z = -247.627  mm,
	W = 0.000 deg,	P = 30.000 deg,	R = 150.585 deg
};
P[154]{
   GP1:
	UF : 0, UT : 1,		CONFIG : 'N U T, 0, 0, 0',
	X = 1249.039  mm,	Y = -257.399  mm,	Z = -247.859  mm,
	W = 0.000 deg,	P = 30.000 deg,	R = 158.269 deg
};
P[155]{
   GP1:
	UF : 0, UT : 1,		CONFIG : 'N U T, 0, 0, 0',
	X = 1250.267  mm,	Y = -255.838  mm,	Z = -248.091  mm,
	W = 0.000 deg,	P = 30.000 deg,	R = 165.953 deg
};
P[156]{
   GP1:
	UF : 0, UT : 1,		CONFIG : 'N U T, 0, 0, 0',
	X = 1251.495  mm,	Y = -254.276  mm,	Z = -248.323  mm,
	W = 0.000 deg,	P = 30.000 deg,	R = 173.637 deg
};
P[157]{
   GP1:
	UF : 0, UT : 1,		CONFIG : 'N U T, 0, 0, 0',
	X = 1252.724  mm,	Y = -252.715  mm,	Z = -248.554  mm,
	W = 0.000 deg,	P = 30.000 deg,	R = -179.771 deg
};
P[158]{
   GP1:
	UF : 0, UT : 1,		CONFIG : 'N U T, 0, 0, 0',
	X = 1253.729  mm,	Y = -250.992  mm,	Z = -248.639  mm,
	W = 0.000 deg,	P = 30.000 deg,	R = -179.771 deg
};
P[159]{
   GP1:
	UF : 0, UT : 1,		CONFIG : 'N U T, 0, 0, 0',
	X = 1247.807  mm,	Y = -249.032  mm,	Z = -248.614  mm,
	W = 0.000 deg,	P = 30.000 deg,	R = -179.771 deg
};
P[160]{
   GP1:
	UF : 0, UT : 1,		CONFIG : 'N U T, 0, 0, 0',
	X = 1253.799  mm,	Y = -247.008  mm,	Z = -248.574  mm,
	W = 0.000 deg,	P = 30.000 deg,	R = -179.771 deg
};
P[161]{
   GP1:
	UF : 0, UT : 1,		CONFIG : 'N U T, 0, 0, 0',
	X = 1253.791  mm,	Y = -245.008  mm,	Z = -248.535  mm,
	W = 0.000 deg,	P = 30.000 deg,	R = -179.771 deg
};
P[162]{
   GP1:
	UF : 0, UT : 1,		CONFIG : 'N U T, 0, 0, 0',
	X = 1253.783  mm,	Y = -243.009  mm,	Z = -248.496  mm,
	W = 0.000 deg,	P = 30.000 deg,	R = -179.771 deg
};
P[163]{
   GP1:
	UF : 0, UT : 1,		CONFIG : 'N U T, 0, 0, 0',
	X = 1253.775  mm,	Y = -241.009  mm,	Z = -248.457  mm,
	W = 0.000 deg,	P = 30.000 deg,	R = -179.771 deg
};
P[164]{
   GP1:
	UF : 0, UT : 1,		CONFIG : 'N U T, 0, 0, 0',
	X = 1247.767  mm,	Y = -239.034  mm,	Z = -248.418  mm,
	W = 0.000 deg,	P = 30.000 deg,	R = -179.771 deg
};
P[165]{
   GP1:
	UF : 0, UT : 1,		CONFIG : 'N U T, 0, 0, 0',
	X = 1247.759  mm,	Y = -237.034  mm,	Z = -248.378  mm,
	W = 0.000 deg,	P = 30.000 deg,	R = -179.771 deg
};
P[166]{
   GP1:
	UF : 0, UT : 1,		CONFIG : 'N U T, 0, 0, 0',
	X = 1253.751  mm,	Y = -235.010  mm,	Z = -248.339  mm,
	W = 0.000 deg,	P = 30.000 deg,	R = -179.771 deg
};
P[167]{
   GP1:
	UF : 0, UT : 1,		CONFIG : 'N U T, 0, 0, 0',
	X = 1253.743  mm,	Y = -233.011  mm,	Z = -248.300  mm,
	W = 0.000 deg,	P = 30.000 deg,	R = -179.771 deg
};
P[168]{
   GP1:
	UF : 0, UT : 1,		CONFIG : 'N U T, 0, 0, 0',
	X = 1253.735  mm,	Y = -231.011  mm,	Z = -248.261  mm,
	W = 0.000 deg,	P = 30.000 deg,	R = -179.771 deg
};
P[169]{
   GP1:
	UF : 0, UT : 1,		CONFIG : 'N U T, 0, 0, 0',
	X = 1253.727  mm,	Y = -229.012  mm,	Z = -248.222  mm,
	W = 0.000 deg,	P = 30.000 deg,	R = -179.771 deg
};
P[170]{
   GP1:
	UF : 0, UT : 1,		CONFIG : 'N U T, 0, 0, 0',
	X = 1253.719  mm,	Y = -227.012  mm,	Z = -248.182  mm,
	W = 0.000 deg,	P = 30.000 deg,	R = -179.771 deg
};
P[171]{
   GP1:
	UF : 0, UT : 1,		CONFIG : 'N U T, 0, 0, 0',
	X = 1253.711  mm,	Y = -225.012  mm,	Z = -248.143  mm,
	W = 0.000 deg,	P = 30.000 deg,	R = -179.771 deg
};
P[172]{
   GP1:
	UF : 0, UT : 1,		CONFIG : 'N U T, 0, 0, 0',
	X = 1247.703  mm,	Y = -223.037  mm,	Z = -248.104  mm,
	W = 0.000 deg,	P = 30.000 deg,	R = -179.771 deg
};
P[173]{
   GP1:
	UF : 0, UT : 1,		CONFIG : 'N U T, 0, 0, 0',
	X = 1247.695  mm,	Y = -221.037  mm,	Z = -248.065  mm,
	W = 0.000 deg,	P = 30.000 deg,	R = -179.771 deg
};
P[174]{
   GP1:
	UF : 0, UT : 1,		CONFIG : 'N U T, 0, 0, 0',
	X = 1253.687  mm,	Y = -219.014  mm,	Z = -248.026  mm,
	W = 0.000 deg,	P = 30.000 deg,	R = -179.771 deg
};
P[175]{
   GP1:
	UF : 0, UT : 1,		CONFIG : 'N U T, 0, 0, 0',
	X = 1253.679  mm,	Y = -217.014  mm,	Z = -247.986  mm,
	W = 0.000 deg,	P = 30.000 deg,	R = -179.771 deg
};
P[176]{
   GP1:
	UF : 0, UT : 1,		CONFIG : 'N U T, 0, 0, 0',
	X = 1253.671  mm,	Y = -215.014  mm,	Z = -247.947  mm,
	W = 0.000 deg,	P = 30.000 deg,	R = -179.771 deg
};
P[177]{
   GP1:
	UF : 0, UT : 1,		CONFIG : 'N U T, 0, 0, 0',
	X = 1253.663  mm,	Y = -213.015  mm,	Z = -247.908  mm,
	W = 0.000 deg,	P = 30.000 deg,	R = -179.771 deg
};
P[178]{
   GP1:
	UF : 0, UT : 1,		CONFIG : 'N U T, 0, 0, 0',
	X = 1253.655  mm,	Y = -211.015  mm,	Z = -247.869  mm,
	W = 0.000 deg,	P = 30.000 deg,	R = -179.771 deg
};
P[179]{
   GP1:
	UF : 0, UT : 1,		CONFIG : 'N U T, 0, 0, 0',
	X = 1247.647  mm,	Y = -209.040  mm,	Z = -247.830  mm,
	W = 0.000 deg,	P = 30.000 deg,	R = -179.771 deg
};
P[180]{
   GP1:
	UF : 0, UT : 1,		CONFIG : 'N U T, 0, 0, 0',
	X = 1247.639  mm,	Y = -207.040  mm,	Z = -247.791  mm,
	W = 0.000 deg,	P = 30.000 deg,	R = -179.771 deg
};
P[181]{
   GP1:
	UF : 0, UT : 1,		CONFIG : 'N U T, 0, 0, 0',
	X = 1253.630  mm,	Y = -205.016  mm,	Z = -247.751  mm,
	W = 0.000 deg,	P = 30.000 deg,	R = -179.771 deg
};
P[182]{
   GP1:
	UF : 0, UT : 1,		CONFIG : 'N U T, 0, 0, 0',
	X = 1253.622  mm,	Y = -203.017  mm,	Z = -247.712  mm,
	W = 0.000 deg,	P = 30.000 deg,	R = -179.771 deg
};
P[183]{
   GP1:
	UF : 0, UT : 1,		CONFIG : 'N U T, 0, 0, 0',
	X = 1253.614  mm,	Y = -201.017  mm,	Z = -247.673  mm,
	W = 0.000 deg,	P = 30.000 deg,	R = -179.771 deg
};
P[184]{
   GP1:
	UF : 0, UT : 1,		CONFIG : 'N U T, 0, 0, 0',
	X = 1253.606  mm,	Y = -199.018  mm,	Z = -247.634  mm,
	W = 0.000 deg,	P = 30.000 deg,	R = -179.771 deg
};
P[185]{
   GP1:
	UF : 0, UT : 1,		CONFIG : 'N U T, 0, 0, 0',
	X = 1253.598  mm,	Y = -197.018  mm,	Z = -247.595  mm,
	W = 0.000 deg,	P = 30.000 deg,	R = -179.771 deg
};
P[186]{
   GP1:
	UF : 0, UT : 1,		CONFIG : 'N U T, 0, 0, 0',
	X = 1247.591  mm,	Y = -195.042  mm,	Z = -247.555  mm,
	W = 0.000 deg,	P = 30.000 deg,	R = -179.771 deg
};
P[187]{
   GP1:
	UF : 0, UT : 1,		CONFIG : 'N U T, 0, 0, 0',
	X = 1247.583  mm,	Y = -193.043  mm,	Z = -247.516  mm,
	W = 0.000 deg,	P = 30.000 deg,	R = -179.771 deg
};
P[188]{
   GP1:
	UF : 0, UT : 1,		CONFIG : 'N U T, 0, 0, 0',
	X = 1253.574  mm,	Y = -191.019  mm,	Z = -247.477  mm,
	W = 0.000 deg,	P = 30.000 deg,	R = -174.933 deg
};
P[189]{
   GP1:
	UF : 0, UT : 1,		CONFIG : 'N U T, 0, 0, 0',
	X = 1253.566  mm,	Y = -189.020  mm,	Z = -247.438  mm,
	W = 0.000 deg,	P = 30.000 deg,	R = -167.339 deg
};
P[190]{
   GP1:
	UF : 0, UT : 1,		CONFIG : 'N U T, 0, 0, 0',
	X = 1253.558  mm,	Y = -187.020  mm,	Z = -247.399  mm,
	W = 0.000 deg,	P = 30.000 deg,	R = -159.745 deg
};
P[191]{
   GP1:
	UF : 0, UT : 1,		CONFIG : 'N U T, 0, 0, 0',
	X = 1253.550  mm,	Y = -185.020  mm,	Z = -247.359  mm,
	W = 0.000 deg,	P = 30.000 deg,	R = -152.151 deg
};
P[192]{
   GP1:
	UF : 0, UT : 1,		CONFIG : 'N U T, 0, 0, 0',
	X = 1253.542  mm,	Y = -183.021  mm,	Z = -247.320  mm,
	W = 0.000 deg,	P = 30.000 deg,	R = -144.557 deg
};
P[193]{
   GP1:
	UF : 0, UT : 1,		CONFIG : 'N U T, 0, 0, 0',
	X = 1253.388  mm,	Y = -181.049  mm,	Z = -247.300  mm,
	W = 0.000 deg,	P = 30.000 deg,	R = -141.800 deg
};
P[194]{
   GP1:
	UF : 0, UT : 1,		CONFIG : 'N U T, 0, 0, 0',
	X = 1247.597  mm,	Y = -183.098  mm,	Z = -247.175  mm,
	W = 0.000 deg,	P = 30.000 deg,	R = -141.800 deg
};
P[195]{
   GP1:
	UF : 0, UT : 1,		CONFIG : 'N U T, 0, 0, 0',
	X = 1246.371  mm,	Y = -181.540  mm,	Z = -246.913  mm,
	W = 0.000 deg,	P = 30.000 deg,	R = -141.800 deg
};
P[196]{
   GP1:
	UF : 0, UT : 1,		CONFIG : 'N U T, 0, 0, 0',
	X = 1249.860  mm,	Y = -176.272  mm,	Z = -246.651  mm,
	W = 0.000 deg,	P = 30.000 deg,	R = -141.800 deg
};
P[197]{
   GP1:
	UF : 0, UT : 1,		CONFIG : 'N U T, 0, 0, 0',
	X = 1248.634  mm,	Y = -174.713  mm,	Z = -246.390  mm,
	W = 0.000 deg,	P = 30.000 deg,	R = -141.800 deg
};
P[198]{
   GP1:
	UF : 0, UT : 1,		CONFIG : 'N U T, 0, 0, 0',
	X = 1242.692  mm,	Y = -176.866  mm,	Z = -246.128  mm,
	W = 0.000 deg,	P = 30.000 deg,	R = -141.800 deg
};
P[199]{
   GP1:
	UF : 0, UT : 1,		CONFIG : 'N U T, 0, 0, 0',
	X = 1241.466  mm,	Y = -175.307  mm,	Z = -245.866  mm,
	W = 0.000 deg,	P = 30.000 deg,	R = -141.800 deg
};
P[200]{
   GP1:
	UF : 0, UT : 1,		CONFIG : 'N U T, 0, 0, 0',
	X = 1244.955  mm,	Y = -170.039  mm,	Z = -245.604  mm,
	W = 0.000 deg,	P = 30.000 deg,	R = -141.800 deg
};
P[201]{
   GP1:
	UF : 0, UT : 1,		CONFIG : 'N U T, 0, 0, 0',
	X = 1243.729  mm,	Y = -168.481  mm,	Z = -245.342  mm,
	W = 0.000 deg,	P = 30.000 deg,	R = -141.800 deg
};
P[202]{
   GP1:
	UF : 0, UT : 1,		CONFIG : 'N U T, 0, 0, 0',
	X = 1242.503  mm,	Y = -166.922  mm,	Z = -245.080  mm,
	W = 0.000 deg,	P = 30.000 deg,	R = -141.800 deg
};
P[203]{
   GP1:
	UF : 0, UT : 1,		CONFIG : 'N U T, 0, 0, 0',
	X = 1236.562  mm,	Y = -169.075  mm,	Z = -244.819  mm,
	W = 0.000 deg,	P = 30.000 deg,	R = -141.800 deg
};
P[204]{
   GP1:
	UF : 0, UT : 1,		CONFIG : 'N U T, 0, 0, 0',
	X = 1235.335  mm,	Y = -167.516  mm,	Z = -244.557  mm,
	W = 0.000 deg,	P = 30.000 deg,	R = -141.800 deg
};
P[205]{
   GP1:
	UF : 0, UT : 1,		CONFIG : 'N U T, 0, 0, 0',
	X = 1234.109  mm,	Y = -165.958  mm,	Z = -244.295  mm,
	W = 0.000 deg,	P = 30.000 deg,	R = -141.800 deg
};
P[206]{
   GP1:
	UF : 0, UT : 1,		CONFIG : 'N U T, 0, 0, 0',
	X = 1232.883  mm,	Y = -164.400  mm,	Z = -244.033  mm,
	W = 0.000 deg,	P = 30.000 deg,	R = -141.800 deg
};
P[207]{
   GP1:
	UF : 0, UT : 1,		CONFIG : 'N U T, 0, 0, 0',
	X = 1236.372  mm,	Y = -159.131  mm,	Z = -243.771  mm,
	W = 0.000 deg,	P = 30.000 deg,	R = -141.800 deg
};
P[208]{
   GP1:
	UF : 0, UT : 1,		CONFIG : 'N U T, 0, 0, 0',
	X = 1230.431  mm,	Y = -161.284  mm,	Z = -243.509  mm,
	W = 0.000 deg,	P = 30.000 deg,	R = -141.800 deg
};
P[209]{
   GP1:
	UF : 0, UT : 1,		CONFIG : 'N U T, 0, 0, 0',
	X = 1229.205  mm,	Y = -159.725  mm,	Z = -243.247  mm,
	W = 0.000 deg,	P = 30.000 deg,	R = -141.800 deg
};
P[210]{
   GP1:
	UF : 0, UT : 1,		CONFIG : 'N U T, 0, 0, 0',
	X = 1232.694  mm,	Y = -154.457  mm,	Z = -242.986  mm,
	W = 0.000 deg,	P = 30.000 deg,	R = -141.800 deg
};
P[211]{
   GP1:
	UF : 0, UT : 1,		CONFIG : 'N U T, 0, 0, 0',
	X = 1231.468  mm,	Y = -152.899  mm,	Z = -242.724  mm,
	W = 0.000 deg,	P = 30.000 deg,	R = -141.800 deg
};
P[212]{
   GP1:
	UF : 0, UT : 1,		CONFIG : 'N U T, 0, 0, 0',
	X = 1230.241  mm,	Y = -151.340  mm,	Z = -242.462  mm,
	W = 0.000 deg,	P = 30.000 deg,	R = -141.800 deg
};
P[213]{
   GP1:
	UF : 0, UT : 1,		CONFIG : 'N U T, 0, 0, 0',
	X = 1229.015  mm,	Y = -149.782  mm,	Z = -242.200  mm,
	W = 0.000 deg,	P = 30.000 deg,	R = -141.800 deg
};
P[214]{
   GP1:
	UF : 0, UT : 1,		CONFIG : 'N U T, 0, 0, 0',
	X = 1223.074  mm,	Y = -151.935  mm,	Z = -241.938  mm,
	W = 0.000 deg,	P = 30.000 deg,	R = -141.800 deg
};
P[215]{
   GP1:
	UF : 0, UT : 1,		CONFIG : 'N U T, 0, 0, 0',
	X = 1221.848  mm,	Y = -150.376  mm,	Z = -241.676  mm,
	W = 0.000 deg,	P = 30.000 deg,	R = -141.800 deg
};
P[216]{
   GP1:
	UF : 0, UT : 1,		CONFIG : 'N U T, 0, 0, 0',
	X = 1220.622  mm,	Y = -148.818  mm,	Z = -241.415  mm,
	W = 0.000 deg,	P = 30.000 deg,	R = -141.800 deg
};
P[217]{
   GP1:
	UF : 0, UT : 1,		CONFIG : 'N U T, 0, 0, 0',
	X = 1219.395  mm,	Y = -147.260  mm,	Z = -241.153  mm,
	W = 0.000 deg,	P = 30.000 deg,	R = -153.708 deg
};
P[218]{
   GP1:
	UF : 0, UT : 1,		CONFIG : 'N U T, 0, 0, 0',
	X = 1218.169  mm,	Y = -145.702  mm,	Z = -240.891  mm,
	W = 0.000 deg,	P = 30.000 deg,	R = -161.776 deg
};
P[219]{
   GP1:
	UF : 0, UT : 1,		CONFIG : 'N U T, 0, 0, 0',
	X = 1216.943  mm,	Y = -144.144  mm,	Z = -240.629  mm,
	W = 0.000 deg,	P = 30.000 deg,	R = -169.844 deg
};
P[220]{
   GP1:
	UF : 0, UT : 1,		CONFIG : 'N U T, 0, 0, 0',
	X = 1215.717  mm,	Y = -142.585  mm,	Z = -240.367  mm,
	W = 0.000 deg,	P = 30.000 deg,	R = -177.911 deg
};
P[221]{
   GP1:
	UF : 0, UT : 1,		CONFIG : 'N U T, 0, 0, 0',
	X = 1214.491  mm,	Y = -141.027  mm,	Z = -240.105  mm,
	W = 0.000 deg,	P = 30.000 deg,	R = 177.861 deg
};
P[222]{
   GP1:
	UF : 0, UT : 1,		CONFIG : 'N U T, 0, 0, 0',
	X = 1213.456  mm,	Y = -139.252  mm,	Z = -240.005  mm,
	W = 0.000 deg,	P = 30.000 deg,	R = 177.861 deg
};
P[223]{
   GP1:
	UF : 0, UT : 1,		CONFIG : 'N U T, 0, 0, 0',
	X = 1213.427  mm,	Y = -137.230  mm,	Z = -239.993  mm,
	W = 0.000 deg,	P = 30.000 deg,	R = 177.861 deg
};
P[224]{
   GP1:
	UF : 0, UT : 1,		CONFIG : 'N U T, 0, 0, 0',
	X = 1213.501  mm,	Y = -135.232  mm,	Z = -239.973  mm,
	W = 0.000 deg,	P = 30.000 deg,	R = 177.861 deg
};
P[225]{
   GP1:
	UF : 0, UT : 1,		CONFIG : 'N U T, 0, 0, 0',
	X = 1213.576  mm,	Y = -133.233  mm,	Z = -239.953  mm,
	W = 0.000 deg,	P = 30.000 deg,	R = 177.861 deg
};
P[226]{
   GP1:
	UF : 0, UT : 1,		CONFIG : 'N U T, 0, 0, 0',
	X = 1213.651  mm,	Y = -131.235  mm,	Z = -239.933  mm,
	W = 0.000 deg,	P = 30.000 deg,	R = 177.861 deg
};
P[227]{
   GP1:
	UF : 0, UT : 1,		CONFIG : 'N U T, 0, 0, 0',
	X = 1219.721  mm,	Y = -129.460  mm,	Z = -239.913  mm,
	W = 0.000 deg,	P = 30.000 deg,	R = 177.861 deg
};
P[228]{
   GP1:
	UF : 0, UT : 1,		CONFIG : 'N U T, 0, 0, 0',
	X = 1213.800  mm,	Y = -127.238  mm,	Z = -239.893  mm,
	W = 0.000 deg,	P = 30.000 deg,	R = 177.861 deg
};
P[229]{
   GP1:
	UF : 0, UT : 1,		CONFIG : 'N U T, 0, 0, 0',
	X = 1213.875  mm,	Y = -125.239  mm,	Z = -239.873  mm,
	W = 0.000 deg,	P = 30.000 deg,	R = 177.861 deg
};
P[230]{
   GP1:
	UF : 0, UT : 1,		CONFIG : 'N U T, 0, 0, 0',
	X = 1213.949  mm,	Y = -123.241  mm,	Z = -239.853  mm,
	W = 0.000 deg,	P = 30.000 deg,	R = 177.861 deg
};
P[231]{
   GP1:
	UF : 0, UT : 1,		CONFIG : 'N U T, 0, 0, 0',
	X = 1214.024  mm,	Y = -121.242  mm,	Z = -239.833  mm,
	W = 0.000 deg,	P = 30.000 deg,	R = 177.861 deg
};
P[232]{
   GP1:
	UF : 0, UT : 1,		CONFIG : 'N U T, 0, 0, 0',
	X = 1220.094  mm,	Y = -119.467  mm,	Z = -239.813  mm,
	W = 0.000 deg,	P = 30.000 deg,	R = 177.861 deg
};
P[233]{
   GP1:
	UF : 0, UT : 1,		CONFIG : 'N U T, 0, 0, 0',
	X = 1214.173  mm,	Y = -117.245  mm,	Z = -239.793  mm,
	W = 0.000 deg,	P = 30.000 deg,	R = 177.861 deg
};
P[234]{
   GP1:
	UF : 0, UT : 1,		CONFIG : 'N U T, 0, 0, 0',
	X = 1214.248  mm,	Y = -115.247  mm,	Z = -239.773  mm,
	W = 0.000 deg,	P = 30.000 deg,	R = 177.861 deg
};
P[235]{
   GP1:
	UF : 0, UT : 1,		CONFIG : 'N U T, 0, 0, 0',
	X = 1214.322  mm,	Y = -113.248  mm,	Z = -239.753  mm,
	W = 0.000 deg,	P = 30.000 deg,	R = 177.861 deg
};
P[236]{
   GP1:
	UF : 0, UT : 1,		CONFIG : 'N U T, 0, 0, 0',
	X = 1214.397  mm,	Y = -111.250  mm,	Z = -239.733  mm,
	W = 0.000 deg,	P = 30.000 deg,	R = 177.861 deg
};
P[237]{
   GP1:
	UF : 0, UT : 1,		CONFIG : 'N U T, 0, 0, 0',
	X = 1220.467  mm,	Y = -109.475  mm,	Z = -239.713  mm,
	W = 0.000 deg,	P = 30.000 deg,	R = 177.861 deg
};
P[238]{
   GP1:
	UF : 0, UT : 1,		CONFIG : 'N U T, 0, 0, 0',
	X = 1214.546  mm,	Y = -107.253  mm,	Z = -239.693  mm,
	W = 0.000 deg,	P = 30.000 deg,	R = 177.861 deg
};
P[239]{
   GP1:
	UF : 0, UT : 1,		CONFIG : 'N U T, 0, 0, 0',
	X = 1214.621  mm,	Y = -105.254  mm,	Z = -239.673  mm,
	W = 0.000 deg,	P = 30.000 deg,	R = 177.861 deg
};
P[240]{
   GP1:
	UF : 0, UT : 1,		CONFIG : 'N U T, 0, 0, 0',
	X = 1220.691  mm,	Y = -103.479  mm,	Z = -239.653  mm,
	W = 0.000 deg,	P = 30.000 deg,	R = 177.861 deg
};
P[241]{
   GP1:
	UF : 0, UT : 1,		CONFIG : 'N U T, 0, 0, 0',
	X = 1214.770  mm,	Y = -101.257  mm,	Z = -239.633  mm,
	W = 0.000 deg,	P = 30.000 deg,	R = 177.861 deg
};
P[242]{
   GP1:
	UF : 0, UT : 1,		CONFIG : 'N U T, 0, 0, 0',
	X = 1214.845  mm,	Y = -99.258  mm,	Z = -239.613  mm,
	W = 0.000 deg,	P = 30.000 deg,	R = 177.861 deg
};
P[243]{
   GP1:
	UF : 0, UT : 1,		CONFIG : 'N U T, 0, 0, 0',
	X = 1214.919  mm,	Y = -97.260  mm,	Z = -239.593  mm,
	W = 0.000 deg,	P = 30.000 deg,	R = 177.861 deg
};
P[244]{
   GP1:
	UF : 0, UT : 1,		CONFIG : 'N U T, 0, 0, 0',
	X = 1214.994  mm,	Y = -95.261  mm,	Z = -239.573  mm,
	W = 0.000 deg,	P = 30.000 deg,	R = 177.861 deg
};
P[245]{
   GP1:
	UF : 0, UT : 1,		CONFIG : 'N U T, 0, 0, 0',
	X = 1221.065  mm,	Y = -93.487  mm,	Z = -239.553  mm,
	W = 0.000 deg,	P = 30.000 deg,	R = 177.861 deg
};
P[246]{
   GP1:
	UF : 0, UT : 1,		CONFIG : 'N U T, 0, 0, 0',
	X = 1215.143  mm,	Y = -91.264  mm,	Z = -239.533  mm,
	W = 0.000 deg,	P = 30.000 deg,	R = 177.861 deg
};
P[247]{
   GP1:
	UF : 0, UT : 1,		CONFIG : 'N U T, 0, 0, 0',
	X = 1215.218  mm,	Y = -89.266  mm,	Z = -239.513  mm,
	W = 0.000 deg,	P = 30.000 deg,	R = 177.861 deg
};
P[248]{
   GP1:
	UF : 0, UT : 1,		CONFIG : 'N U T, 0, 0, 0',
	X = 1215.293  mm,	Y = -87.267  mm,	Z = -239.493  mm,
	W = 0.000 deg,	P = 30.000 deg,	R = 177.861 deg
};
P[249]{
   GP1:
	UF : 0, UT : 1,		CONFIG : 'N U T, 0, 0, 0',
	X = 1215.367  mm,	Y = -85.269  mm,	Z = -239.473  mm,
	W = 0.000 deg,	P = 30.000 deg,	R = 177.861 deg
};
P[250]{
   GP1:
	UF : 0, UT : 1,		CONFIG : 'N U T, 0, 0, 0',
	X = 1221.438  mm,	Y = -83.494  mm,	Z = -239.453  mm,
	W = 0.000 deg,	P = 30.000 deg,	R = 177.861 deg
};
P[251]{
   GP1:
	UF : 0, UT : 1,		CONFIG : 'N U T, 0, 0, 0',
	X = 1215.516  mm,	Y = -81.272  mm,	Z = -239.433  mm,
	W = 0.000 deg,	P = 30.000 deg,	R = 177.861 deg
};
P[252]{
   GP1:
	UF : 0, UT : 1,		CONFIG : 'N U T, 0, 0, 0',
	X = 1215.591  mm,	Y = -79.273  mm,	Z = -239.413  mm,
	W = 0.000 deg,	P = 30.000 deg,	R = 177.861 deg
};
P[253]{
   GP1:
	UF : 0, UT : 1,		CONFIG : 'N U T, 0, 0, 0',
	X = 1215.666  mm,	Y = -77.275  mm,	Z = -239.393  mm,
	W = 0.000 deg,	P = 30.000 deg,	R = 177.861 deg
};
P[254]{
   GP1:
	UF : 0, UT : 1,		CONFIG : 'N U T, 0, 0, 0',
	X = 1215.740  mm,	Y = -75.276  mm,	Z = -239.373  mm,
	W = 0.000 deg,	P = 30.000 deg,	R = 165.611 deg
};
P[255]{
   GP1:
	UF : 0, UT : 1,		CONFIG : 'N U T, 0, 0, 0',
	X = 1215.815  mm,	Y = -73.278  mm,	Z = -239.353  mm,
	W = 0.000 deg,	P = 30.000 deg,	R = 158.034 deg
};
P[256]{
   GP1:
	UF : 0, UT : 1,		CONFIG : 'N U T, 0, 0, 0',
	X = 1215.890  mm,	Y = -71.279  mm,	Z = -239.333  mm,
	W = 0.000 deg,	P = 30.000 deg,	R = 150.458 deg
};
P[257]{
   GP1:
	UF : 0, UT : 1,		CONFIG : 'N U T, 0, 0, 0',
	X = 1215.964  mm,	Y = -69.281  mm,	Z = -239.313  mm,
	W = 0.000 deg,	P = 30.000 deg,	R = 142.881 deg
};
P[258]{
   GP1:
	UF : 0, UT : 1,		CONFIG : 'N U T, 0, 0, 0',
	X = 1216.039  mm,	Y = -67.282  mm,	Z = -239.293  mm,
	W = 0.000 deg,	P = 30.000 deg,	R = 139.979 deg
};
P[259]{
   GP1:
	UF : 0, UT : 1,		CONFIG : 'N U T, 0, 0, 0',
	X = 1216.492  mm,	Y = -65.365  mm,	Z = -239.288  mm,
	W = 0.000 deg,	P = 30.000 deg,	R = 139.979 deg
};
P[260]{
   GP1:
	UF : 0, UT : 1,		CONFIG : 'N U T, 0, 0, 0',
	X = 1222.327  mm,	Y = -67.691  mm,	Z = -239.482  mm,
	W = 0.000 deg,	P = 30.000 deg,	R = 139.979 deg
};
P[261]{
   GP1:
	UF : 0, UT : 1,		CONFIG : 'N U T, 0, 0, 0',
	X = 1223.603  mm,	Y = -66.172  mm,	Z = -239.735  mm,
	W = 0.000 deg,	P = 30.000 deg,	R = 139.979 deg
};
P[262]{
   GP1:
	UF : 0, UT : 1,		CONFIG : 'N U T, 0, 0, 0',
	X = 1224.879  mm,	Y = -64.653  mm,	Z = -239.987  mm,
	W = 0.000 deg,	P = 30.000 deg,	R = 139.979 deg
};
P[263]{
   GP1:
	UF : 0, UT : 1,		CONFIG : 'N U T, 0, 0, 0',
	X = 1226.155  mm,	Y = -63.134  mm,	Z = -240.240  mm,
	W = 0.000 deg,	P = 30.000 deg,	R = 139.979 deg
};
P[264]{
   GP1:
	UF : 0, UT : 1,		CONFIG : 'N U T, 0, 0, 0',
	X = 1227.431  mm,	Y = -61.614  mm,	Z = -240.493  mm,
	W = 0.000 deg,	P = 30.000 deg,	R = 139.979 deg
};
P[265]{
   GP1:
	UF : 0, UT : 1,		CONFIG : 'N U T, 0, 0, 0',
	X = 1224.112  mm,	Y = -56.236  mm,	Z = -240.746  mm,
	W = 0.000 deg,	P = 30.000 deg,	R = 139.979 deg
};
P[266]{
   GP1:
	UF : 0, UT : 1,		CONFIG : 'N U T, 0, 0, 0',
	X = 1225.388  mm,	Y = -54.717  mm,	Z = -240.999  mm,
	W = 0.000 deg,	P = 30.000 deg,	R = 139.979 deg
};
P[267]{
   GP1:
	UF : 0, UT : 1,		CONFIG : 'N U T, 0, 0, 0',
	X = 1231.258  mm,	Y = -57.056  mm,	Z = -241.252  mm,
	W = 0.000 deg,	P = 30.000 deg,	R = 139.979 deg
};
P[268]{
   GP1:
	UF : 0, UT : 1,		CONFIG : 'N U T, 0, 0, 0',
	X = 1232.534  mm,	Y = -55.537  mm,	Z = -241.504  mm,
	W = 0.000 deg,	P = 30.000 deg,	R = 139.979 deg
};
P[269]{
   GP1:
	UF : 0, UT : 1,		CONFIG : 'N U T, 0, 0, 0',
	X = 1233.810  mm,	Y = -54.018  mm,	Z = -241.757  mm,
	W = 0.000 deg,	P = 30.000 deg,	R = 139.979 deg
};
P[270]{
   GP1:
	UF : 0, UT : 1,		CONFIG : 'N U T, 0, 0, 0',
	X = 1235.086  mm,	Y = -52.498  mm,	Z = -242.010  mm,
	W = 0.000 deg,	P = 30.000 deg,	R = 139.979 deg
};
P[271]{
   GP1:
	UF : 0, UT : 1,		CONFIG : 'N U T, 0, 0, 0',
	X = 1231.767  mm,	Y = -47.120  mm,	Z = -242.263  mm,
	W = 0.000 deg,	P = 30.000 deg,	R = 139.979 deg
};
P[272]{
   GP1:
	UF : 0, UT : 1,		CONFIG : 'N U T, 0, 0, 0',
	X = 1233.043  mm,	Y = -45.601  mm,	Z = -242.516  mm,
	W = 0.000 deg,	P = 30.000 deg,	R = 139.979 deg
};
P[273]{
   GP1:
	UF : 0, UT : 1,		CONFIG : 'N U T, 0, 0, 0',
	X = 1238.913  mm,	Y = -47.940  mm,	Z = -242.769  mm,
	W = 0.000 deg,	P = 30.000 deg,	R = 139.979 deg
};
P[274]{
   GP1:
	UF : 0, UT : 1,		CONFIG : 'N U T, 0, 0, 0',
	X = 1240.189  mm,	Y = -46.421  mm,	Z = -243.021  mm,
	W = 0.000 deg,	P = 30.000 deg,	R = 139.979 deg
};
P[275]{
   GP1:
	UF : 0, UT : 1,		CONFIG : 'N U T, 0, 0, 0',
	X = 1241.465  mm,	Y = -44.902  mm,	Z = -243.274  mm,
	W = 0.000 deg,	P = 30.000 deg,	R = 139.979 deg
};
P[276]{
   GP1:
	UF : 0, UT : 1,		CONFIG : 'N U T, 0, 0, 0',
	X = 1242.741  mm,	Y = -43.382  mm,	Z = -243.527  mm,
	W = 0.000 deg,	P = 30.000 deg,	R = 139.979 deg
};
P[277]{
   GP1:
	UF : 0, UT : 1,		CONFIG : 'N U T, 0, 0, 0',
	X = 1244.016  mm,	Y = -41.863  mm,	Z = -243.780  mm,
	W = 0.000 deg,	P = 30.000 deg,	R = 139.979 deg
};
P[278]{
   GP1:
	UF : 0, UT : 1,		CONFIG : 'N U T, 0, 0, 0',
	X = 1240.697  mm,	Y = -36.485  mm,	Z = -244.033  mm,
	W = 0.000 deg,	P = 30.000 deg,	R = 139.979 deg
};
P[279]{
   GP1:
	UF : 0, UT : 1,		CONFIG : 'N U T, 0, 0, 0',
	X = 1241.973  mm,	Y = -34.966  mm,	Z = -244.286  mm,
	W = 0.000 deg,	P = 30.000 deg,	R = 139.979 deg
};
P[280]{
   GP1:
	UF : 0, UT : 1,		CONFIG : 'N U T, 0, 0, 0',
	X = 1247.844  mm,	Y = -37.305  mm,	Z = -244.538  mm,
	W = 0.000 deg,	P = 30.000 deg,	R = 139.979 deg
};
P[281]{
   GP1:
	UF : 0, UT : 1,		CONFIG : 'N U T, 0, 0, 0',
	X = 1249.120  mm,	Y = -35.786  mm,	Z = -244.791  mm,
	W = 0.000 deg,	P = 30.000 deg,	R = 139.979 deg
};
P[282]{
   GP1:
	UF : 0, UT : 1,		CONFIG : 'N U T, 0, 0, 0',
	X = 1250.396  mm,	Y = -34.266  mm,	Z = -245.044  mm,
	W = 0.000 deg,	P = 30.000 deg,	R = 146.112 deg
};
P[283]{
   GP1:
	UF : 0, UT : 1,		CONFIG : 'N U T, 0, 0, 0',
	X = 1251.671  mm,	Y = -32.747  mm,	Z = -245.297  mm,
	W = 0.000 deg,	P = 30.000 deg,	R = 154.132 deg
};
P[284]{
   GP1:
	UF : 0, UT : 1,		CONFIG : 'N U T, 0, 0, 0',
	X = 1252.947  mm,	Y = -31.228  mm,	Z = -245.550  mm,
	W = 0.000 deg,	P = 30.000 deg,	R = 162.151 deg
};
P[285]{
   GP1:
	UF : 0, UT : 1,		CONFIG : 'N U T, 0, 0, 0',
	X = 1254.223  mm,	Y = -29.708  mm,	Z = -245.802  mm,
	W = 0.000 deg,	P = 30.000 deg,	R = 170.171 deg
};
P[286]{
   GP1:
	UF : 0, UT : 1,		CONFIG : 'N U T, 0, 0, 0',
	X = 1255.499  mm,	Y = -28.189  mm,	Z = -246.055  mm,
	W = 0.000 deg,	P = 30.000 deg,	R = 178.190 deg
};
P[287]{
   GP1:
	UF : 0, UT : 1,		CONFIG : 'N U T, 0, 0, 0',
	X = 1256.767  mm,	Y = -26.661  mm,	Z = -246.275  mm,
	W = 0.000 deg,	P = 30.000 deg,	R = -179.923 deg
};
P[288]{
   GP1:
	UF : 0, UT : 1,		CONFIG : 'N U T, 0, 0, 0',
	X = 1257.312  mm,	Y = -24.674  mm,	Z = -246.272  mm,
	W = 0.000 deg,	P = 30.000 deg,	R = -179.923 deg
};
P[289]{
   GP1:
	UF : 0, UT : 1,		CONFIG : 'N U T, 0, 0, 0',
	X = 1257.309  mm,	Y = -22.674  mm,	Z = -246.247  mm,
	W = 0.000 deg,	P = 30.000 deg,	R = -179.923 deg
};
P[290]{
   GP1:
	UF : 0, UT : 1,		CONFIG : 'N U T, 0, 0, 0',
	X = 1251.307  mm,	Y = -20.683  mm,	Z = -246.223  mm,
	W = 0.000 deg,	P = 30.000 deg,	R = -179.923 deg
};
P[291]{
   GP1:
	UF : 0, UT : 1,		CONFIG : 'N U T, 0, 0, 0',
	X = 1251.304  mm,	Y = -18.683  mm,	Z = -246.198  mm,
	W = 0.000 deg,	P = 30.000 deg,	R = -179.923 deg
};
P[292]{
   GP1:
	UF : 0, UT : 1,		CONFIG : 'N U T, 0, 0, 0',
	X = 1257.301  mm,	Y = -16.675  mm,	Z = -246.173  mm,
	W = 0.000 deg,	P = 30.000 deg,	R = -179.923 deg
};
P[293]{
   GP1:
	UF : 0, UT : 1,		CONFIG : 'N U T, 0, 0, 0',
	X = 1251.299  mm,	Y = -14.683  mm,	Z = -246.149  mm,
	W = 0.000 deg,	P = 30.000 deg,	R = -179.923 deg
};
P[294]{
   GP1:
	UF : 0, UT : 1,		CONFIG : 'N U T, 0, 0, 0',
	X = 1251.296  mm,	Y = -12.683  mm,	Z = -246.124  mm,
	W = 0.000 deg,	P = 30.000 deg,	R = -179.923 deg
};
P[295]{
   GP1:
	UF : 0, UT : 1,		CONFIG : 'N U T, 0, 0, 0',
	X = 1257.293  mm,	Y = -10.675  mm,	Z = -246.099  mm,
	W = 0.000 deg,	P = 30.000 deg,	R = -179.923 deg
};
P[296]{
   GP1:
	UF : 0, UT : 1,		CONFIG : 'N U T, 0, 0, 0',
	X = 1257.290  mm,	Y = -8.676  mm,	Z = -246.074  mm,
	W = 0.000 deg,	P = 30.000 deg,	R = -179.923 deg
};
P[297]{
   GP1:
	UF : 0, UT : 1,		CONFIG : 'N U T, 0, 0, 0',
	X = 1251.288  mm,	Y = -6.684  mm,	Z = -246.050  mm,
	W = 0.000 deg,	P = 30.000 deg,	R = -179.923 deg
};
P[298]{
   GP1:
	UF : 0, UT : 1,		CONFIG : 'N U T, 0, 0, 0',
	X = 1251.285  mm,	Y = -4.684  mm,	Z = -246.025  mm,
	W = 0.000 deg,	P = 30.000 deg,	R = -179.923 deg
};
P[299]{
   GP1:
	UF : 0, UT : 1,		CONFIG : 'N U T, 0, 0, 0',
	X = 1257.282  mm,	Y = -2.676  mm,	Z = -246.000  mm,
	W = 0.000 deg,	P = 30.000 deg,	R = -179.923 deg
};
P[300]{
   GP1:
	UF : 0, UT : 1,		CONFIG : 'N U T, 0, 0, 0',
	X = 1251.280  mm,	Y = -0.684  mm,	Z = -245.975  mm,
	W = 0.000 deg,	P = 30.000 deg,	R = -179.923 deg
};
P[301]{
   GP1:
	UF : 0, UT : 1,		CONFIG : 'N U T, 0, 0, 0',
	X = 1251.277  mm,	Y = 1.316  mm,	Z = -245.951  mm,
	W = 0.000 deg,	P = 30.000 deg,	R = -179.923 deg
};
P[302]{
   GP1:
	UF : 0, UT : 1,		CONFIG : 'N U T, 0, 0, 0',
	X = 1257.274  mm,	Y = 3.324  mm,	Z = -245.926  mm,
	W = 0.000 deg,	P = 30.000 deg,	R = -179.923 deg
};
P[303]{
   GP1:
	UF : 0, UT : 1,		CONFIG : 'N U T, 0, 0, 0',
	X = 1251.272  mm,	Y = 5.315  mm,	Z = -245.901  mm,
	W = 0.000 deg,	P = 30.000 deg,	R = -179.923 deg
};
P[304]{
   GP1:
	UF : 0, UT : 1,		CONFIG : 'N U T, 0, 0, 0',
	X = 1251.269  mm,	Y = 7.315  mm,	Z = -245.876  mm,
	W = 0.000 deg,	P = 30.000 deg,	R = -179.923 deg
};
P[305]{
   GP1:
	UF : 0, UT : 1,		CONFIG : 'N U T, 0, 0, 0',
	X = 1257.266  mm,	Y = 9.323  mm,	Z = -245.852  mm,
	W = 0.000 deg,	P = 30.000 deg,	R = -179.923 deg
};
P[306]{
   GP1:
	UF : 0, UT : 1,		CONFIG : 'N U T, 0, 0, 0',
	X = 1257.264  mm,	Y = 11.323  mm,	Z = -245.827  mm,
	W = 0.000 deg,	P = 30.000 deg,	R = -179.923 deg
};
P[307]{
   GP1:
	UF : 0, UT : 1,		CONFIG : 'N U T, 0, 0, 0',
	X = 1251.261  mm,	Y = 13.315  mm,	Z = -245.802  mm,
	W = 0.000 deg,	P = 30.000 deg,	R = -179.923 deg
};
P[308]{
   GP1:
	UF : 0, UT : 1,		CONFIG : 'N U T, 0, 0, 0',
	X = 1251.258  mm,	Y = 15.315  mm,	Z = -245.777  mm,
	W = 0.000 deg,	P = 30.000 deg,	R = -179.923 deg
};
P[309]{
   GP1:
	UF : 0, UT : 1,		CONFIG : 'N U T, 0, 0, 0',
	X = 1257.255  mm,	Y = 17.322  mm,	Z = -245.753  mm,
	W = 0.000 deg,	P = 30.000 deg,	R = -179.923 deg
};
P[310]{
   GP1:
	UF : 0, UT : 1,		CONFIG : 'N U T, 0, 0, 0',
	X = 1251.253  mm,	Y = 19.314  mm,	Z = -245.728  mm,
	W = 0.000 deg,	P = 30.000 deg,	R = -179.923 deg
};
P[311]{
   GP1:
	UF : 0, UT : 1,		CONFIG : 'N U T, 0, 0, 0',
	X = 1251.250  mm,	Y = 21.314  mm,	Z = -245.703  mm,
	W = 0.000 deg,	P = 30.000 deg,	R = -179.923 deg
};
P[312]{
   GP1:
	UF : 0, UT : 1,		CONFIG : 'N U T, 0, 0, 0',
	X = 1257.247  mm,	Y = 23.322  mm,	Z = -245.678  mm,
	W = 0.000 deg,	P = 30.000 deg,	R = -179.923 deg
};
P[313]{
   GP1:
	UF : 0, UT : 1,		CONFIG : 'N U T, 0, 0, 0',
	X = 1251.245  mm,	Y = 25.314  mm,	Z = -245.654  mm,
	W = 0.000 deg,	P = 30.000 deg,	R = -179.923 deg
};
P[314]{
   GP1:
	UF : 0, UT : 1,		CONFIG : 'N U T, 0, 0, 0',
	X = 1251.242  mm,	Y = 27.314  mm,	Z = -245.629  mm,
	W = 0.000 deg,	P = 30.000 deg,	R = -179.923 deg
};
P[315]{
   GP1:
	UF : 0, UT : 1,		CONFIG : 'N U T, 0, 0, 0',
	X = 1257.239  mm,	Y = 29.322  mm,	Z = -245.604  mm,
	W = 0.000 deg,	P = 30.000 deg,	R = -179.923 deg
};
P[316]{
   GP1:
	UF : 0, UT : 1,		CONFIG : 'N U T, 0, 0, 0',
	X = 1257.237  mm,	Y = 31.321  mm,	Z = -245.579  mm,
	W = 0.000 deg,	P = 30.000 deg,	R = -179.923 deg
};
P[317]{
   GP1:
	UF : 0, UT : 1,		CONFIG : 'N U T, 0, 0, 0',
	X = 1251.234  mm,	Y = 33.313  mm,	Z = -245.555  mm,
	W = 0.000 deg,	P = 30.000 deg,	R = -179.923 deg
};
P[318]{
   GP1:
	UF : 0, UT : 1,		CONFIG : 'N U T, 0, 0, 0',
	X = 1257.231  mm,	Y = 35.321  mm,	Z = -245.530  mm,
	W = 0.000 deg,	P = 30.000 deg,	R = -171.534 deg
};
P[319]{
   GP1:
	UF : 0, UT : 1,		CONFIG : 'N U T, 0, 0, 0',
	X = 1257.229  mm,	Y = 37.321  mm,	Z = -245.505  mm,
	W = 0.000 deg,	P = 30.000 deg,	R = -164.106 deg
};
P[320]{
   GP1:
	UF : 0, UT : 1,		CONFIG : 'N U T, 0, 0, 0',
	X = 1257.226  mm,	Y = 39.321  mm,	Z = -245.480  mm,
	W = 0.000 deg,	P = 30.000 deg,	R = -156.678 deg
};
P[321]{
   GP1:
	UF : 0, UT : 1,		CONFIG : 'N U T, 0, 0, 0',
	X = 1257.223  mm,	Y = 41.321  mm,	Z = -245.456  mm,
	W = 0.000 deg,	P = 30.000 deg,	R = -149.250 deg
};
P[322]{
   GP1:
	UF : 0, UT : 1,		CONFIG : 'N U T, 0, 0, 0',
	X = 1257.220  mm,	Y = 43.320  mm,	Z = -245.431  mm,
	W = 0.000 deg,	P = 30.000 deg,	R = -142.783 deg
};
P[323]{
   GP1:
	UF : 0, UT : 1,		CONFIG : 'N U T, 0, 0, 0',
	X = 1256.695  mm,	Y = 45.170  mm,	Z = -245.429  mm,
	W = 0.000 deg,	P = 30.000 deg,	R = -142.783 deg
};
P[324]{
   GP1:
	UF : 0, UT : 1,		CONFIG : 'N U T, 0, 0, 0',
	X = 1255.505  mm,	Y = 46.743  mm,	Z = -245.191  mm,
	W = 0.000 deg,	P = 30.000 deg,	R = -142.783 deg
};
P[325]{
   GP1:
	UF : 0, UT : 1,		CONFIG : 'N U T, 0, 0, 0',
	X = 1254.305  mm,	Y = 48.323  mm,	Z = -244.932  mm,
	W = 0.000 deg,	P = 30.000 deg,	R = -142.783 deg
};
P[326]{
   GP1:
	UF : 0, UT : 1,		CONFIG : 'N U T, 0, 0, 0',
	X = 1248.328  mm,	Y = 46.273  mm,	Z = -244.673  mm,
	W = 0.000 deg,	P = 30.000 deg,	R = -142.783 deg
};
P[327]{
   GP1:
	UF : 0, UT : 1,		CONFIG : 'N U T, 0, 0, 0',
	X = 1251.906  mm,	Y = 51.481  mm,	Z = -244.415  mm,
	W = 0.000 deg,	P = 30.000 deg,	R = -142.783 deg
};
P[328]{
   GP1:
	UF : 0, UT : 1,		CONFIG : 'N U T, 0, 0, 0',
	X = 1250.707  mm,	Y = 53.061  mm,	Z = -244.156  mm,
	W = 0.000 deg,	P = 30.000 deg,	R = -142.783 deg
};
P[329]{
   GP1:
	UF : 0, UT : 1,		CONFIG : 'N U T, 0, 0, 0',
	X = 1244.729  mm,	Y = 51.011  mm,	Z = -243.898  mm,
	W = 0.000 deg,	P = 30.000 deg,	R = -142.783 deg
};
P[330]{
   GP1:
	UF : 0, UT : 1,		CONFIG : 'N U T, 0, 0, 0',
	X = 1248.308  mm,	Y = 56.219  mm,	Z = -243.639  mm,
	W = 0.000 deg,	P = 30.000 deg,	R = -142.783 deg
};
P[331]{
   GP1:
	UF : 0, UT : 1,		CONFIG : 'N U T, 0, 0, 0',
	X = 1247.108  mm,	Y = 57.799  mm,	Z = -243.380  mm,
	W = 0.000 deg,	P = 30.000 deg,	R = -142.783 deg
};
P[332]{
   GP1:
	UF : 0, UT : 1,		CONFIG : 'N U T, 0, 0, 0',
	X = 1245.909  mm,	Y = 59.378  mm,	Z = -243.122  mm,
	W = 0.000 deg,	P = 30.000 deg,	R = -142.783 deg
};
P[333]{
   GP1:
	UF : 0, UT : 1,		CONFIG : 'N U T, 0, 0, 0',
	X = 1244.709  mm,	Y = 60.957  mm,	Z = -242.863  mm,
	W = 0.000 deg,	P = 30.000 deg,	R = -142.783 deg
};
P[334]{
   GP1:
	UF : 0, UT : 1,		CONFIG : 'N U T, 0, 0, 0',
	X = 1238.731  mm,	Y = 58.908  mm,	Z = -242.605  mm,
	W = 0.000 deg,	P = 30.000 deg,	R = -142.783 deg
};
P[335]{
   GP1:
	UF : 0, UT : 1,		CONFIG : 'N U T, 0, 0, 0',
	X = 1242.310  mm,	Y = 64.116  mm,	Z = -242.346  mm,
	W = 0.000 deg,	P = 30.000 deg,	R = -142.783 deg
};
P[336]{
   GP1:
	UF : 0, UT : 1,		CONFIG : 'N U T, 0, 0, 0',
	X = 1241.110  mm,	Y = 65.695  mm,	Z = -242.088  mm,
	W = 0.000 deg,	P = 30.000 deg,	R = -142.783 deg
};
P[337]{
   GP1:
	UF : 0, UT : 1,		CONFIG : 'N U T, 0, 0, 0',
	X = 1235.133  mm,	Y = 63.646  mm,	Z = -241.829  mm,
	W = 0.000 deg,	P = 30.000 deg,	R = -142.783 deg
};
P[338]{
   GP1:
	UF : 0, UT : 1,		CONFIG : 'N U T, 0, 0, 0',
	X = 1238.711  mm,	Y = 68.854  mm,	Z = -241.570  mm,
	W = 0.000 deg,	P = 30.000 deg,	R = -142.783 deg
};
P[339]{
   GP1:
	UF : 0, UT : 1,		CONFIG : 'N U T, 0, 0, 0',
	X = 1237.512  mm,	Y = 70.433  mm,	Z = -241.312  mm,
	W = 0.000 deg,	P = 30.000 deg,	R = -142.783 deg
};
P[340]{
   GP1:
	UF : 0, UT : 1,		CONFIG : 'N U T, 0, 0, 0',
	X = 1231.534  mm,	Y = 68.384  mm,	Z = -241.053  mm,
	W = 0.000 deg,	P = 30.000 deg,	R = -142.783 deg
};
P[341]{
   GP1:
	UF : 0, UT : 1,		CONFIG : 'N U T, 0, 0, 0',
	X = 1235.113  mm,	Y = 73.592  mm,	Z = -240.795  mm,
	W = 0.000 deg,	P = 30.000 deg,	R = -142.783 deg
};
P[342]{
   GP1:
	UF : 0, UT : 1,		CONFIG : 'N U T, 0, 0, 0',
	X = 1233.913  mm,	Y = 75.171  mm,	Z = -240.536  mm,
	W = 0.000 deg,	P = 30.000 deg,	R = -142.783 deg
};
P[343]{
   GP1:
	UF : 0, UT : 1,		CONFIG : 'N U T, 0, 0, 0',
	X = 1227.936  mm,	Y = 73.122  mm,	Z = -240.277  mm,
	W = 0.000 deg,	P = 30.000 deg,	R = -142.783 deg
};
P[344]{
   GP1:
	UF : 0, UT : 1,		CONFIG : 'N U T, 0, 0, 0',
	X = 1231.514  mm,	Y = 78.330  mm,	Z = -240.019  mm,
	W = 0.000 deg,	P = 30.000 deg,	R = -142.783 deg
};
P[345]{
   GP1:
	UF : 0, UT : 1,		CONFIG : 'N U T, 0, 0, 0',
	X = 1230.315  mm,	Y = 79.909  mm,	Z = -239.760  mm,
	W = 0.000 deg,	P = 30.000 deg,	R = -142.783 deg
};
P[346]{
   GP1:
	UF : 0, UT : 1,		CONFIG : 'N U T, 0, 0, 0',
	X = 1229.115  mm,	Y = 81.489  mm,	Z = -239.502  mm,
	W = 0.000 deg,	P = 30.000 deg,	R = -142.783 deg
};
P[347]{
   GP1:
	UF : 0, UT : 1,		CONFIG : 'N U T, 0, 0, 0',
	X = 1227.916  mm,	Y = 83.068  mm,	Z = -239.243  mm,
	W = 0.000 deg,	P = 30.000 deg,	R = -142.783 deg
};
P[348]{
   GP1:
	UF : 0, UT : 1,		CONFIG : 'N U T, 0, 0, 0',
	X = 1221.938  mm,	Y = 81.018  mm,	Z = -238.984  mm,
	W = 0.000 deg,	P = 30.000 deg,	R = -157.927 deg
};
P[349]{
   GP1:
	UF : 0, UT : 1,		CONFIG : 'N U T, 0, 0, 0',
	X = 1220.739  mm,	Y = 82.598  mm,	Z = -238.726  mm,
	W = 0.000 deg,	P = 30.000 deg,	R = -165.810 deg
};
P[350]{
   GP1:
	UF : 0, UT : 1,		CONFIG : 'N U T, 0, 0, 0',
	X = 1219.539  mm,	Y = 84.177  mm,	Z = -238.467  mm,
	W = 0.000 deg,	P = 30.000 deg,	R = -173.693 deg
};
P[351]{
   GP1:
	UF : 0, UT : 1,		CONFIG : 'N U T, 0, 0, 0',
	X = 1218.340  mm,	Y = 85.756  mm,	Z = -238.209  mm,
	W = 0.000 deg,	P = 30.000 deg,	R = 178.423 deg
};
P[352]{
   GP1:
	UF : 0, UT : 1,		CONFIG : 'N U T, 0, 0, 0',
	X = 1217.189  mm,	Y = 87.387  mm,	Z = -238.032  mm,
	W = 0.000 deg,	P = 30.000 deg,	R = 177.800 deg
};
P[353]{
   GP1:
	UF : 0, UT : 1,		CONFIG : 'N U T, 0, 0, 0',
	X = 1222.933  mm,	Y = 89.169  mm,	Z = -238.028  mm,
	W = 0.000 deg,	P = 30.000 deg,	R = 177.800 deg
};
P[354]{
   GP1:
	UF : 0, UT : 1,		CONFIG : 'N U T, 0, 0, 0',
	X = 1217.014  mm,	Y = 91.397  mm,	Z = -238.015  mm,
	W = 0.000 deg,	P = 30.000 deg,	R = 177.800 deg
};
P[355]{
   GP1:
	UF : 0, UT : 1,		CONFIG : 'N U T, 0, 0, 0',
	X = 1223.087  mm,	Y = 93.166  mm,	Z = -238.001  mm,
	W = 0.000 deg,	P = 30.000 deg,	R = 177.800 deg
};
P[356]{
   GP1:
	UF : 0, UT : 1,		CONFIG : 'N U T, 0, 0, 0',
	X = 1223.164  mm,	Y = 95.164  mm,	Z = -237.988  mm,
	W = 0.000 deg,	P = 30.000 deg,	R = 177.800 deg
};
P[357]{
   GP1:
	UF : 0, UT : 1,		CONFIG : 'N U T, 0, 0, 0',
	X = 1223.240  mm,	Y = 97.162  mm,	Z = -237.975  mm,
	W = 0.000 deg,	P = 30.000 deg,	R = 177.800 deg
};
P[358]{
   GP1:
	UF : 0, UT : 1,		CONFIG : 'N U T, 0, 0, 0',
	X = 1223.317  mm,	Y = 99.161  mm,	Z = -237.962  mm,
	W = 0.000 deg,	P = 30.000 deg,	R = 177.800 deg
};
P[359]{
   GP1:
	UF : 0, UT : 1,		CONFIG : 'N U T, 0, 0, 0',
	X = 1223.394  mm,	Y = 101.159  mm,	Z = -237.948  mm,
	W = 0.000 deg,	P = 30.000 deg,	R = 177.800 deg
};
P[360]{
   GP1:
	UF : 0, UT : 1,		CONFIG : 'N U T, 0, 0, 0',
	X = 1223.471  mm,	Y = 103.158  mm,	Z = -237.935  mm,
	W = 0.000 deg,	P = 30.000 deg,	R = 177.800 deg
};
P[361]{
   GP1:
	UF : 0, UT : 1,		CONFIG : 'N U T, 0, 0, 0',
	X = 1223.547  mm,	Y = 105.156  mm,	Z = -237.922  mm,
	W = 0.000 deg,	P = 30.000 deg,	R = 177.800 deg
};
P[362]{
   GP1:
	UF : 0, UT : 1,		CONFIG : 'N U T, 0, 0, 0',
	X = 1223.624  mm,	Y = 107.155  mm,	Z = -237.908  mm,
	W = 0.000 deg,	P = 30.000 deg,	R = 177.800 deg
};
P[363]{
   GP1:
	UF : 0, UT : 1,		CONFIG : 'N U T, 0, 0, 0',
	X = 1223.701  mm,	Y = 109.153  mm,	Z = -237.895  mm,
	W = 0.000 deg,	P = 30.000 deg,	R = 177.800 deg
};
P[364]{
   GP1:
	UF : 0, UT : 1,		CONFIG : 'N U T, 0, 0, 0',
	X = 1223.778  mm,	Y = 111.152  mm,	Z = -237.882  mm,
	W = 0.000 deg,	P = 30.000 deg,	R = 177.800 deg
};
P[365]{
   GP1:
	UF : 0, UT : 1,		CONFIG : 'N U T, 0, 0, 0',
	X = 1223.855  mm,	Y = 113.150  mm,	Z = -237.868  mm,
	W = 0.000 deg,	P = 30.000 deg,	R = 177.800 deg
};
P[366]{
   GP1:
	UF : 0, UT : 1,		CONFIG : 'N U T, 0, 0, 0',
	X = 1223.931  mm,	Y = 115.149  mm,	Z = -237.855  mm,
	W = 0.000 deg,	P = 30.000 deg,	R = 177.800 deg
};
P[367]{
   GP1:
	UF : 0, UT : 1,		CONFIG : 'N U T, 0, 0, 0',
	X = 1224.008  mm,	Y = 117.147  mm,	Z = -237.842  mm,
	W = 0.000 deg,	P = 30.000 deg,	R = 177.800 deg
};
P[368]{
   GP1:
	UF : 0, UT : 1,		CONFIG : 'N U T, 0, 0, 0',
	X = 1224.085  mm,	Y = 119.146  mm,	Z = -237.828  mm,
	W = 0.000 deg,	P = 30.000 deg,	R = 177.800 deg
};
P[369]{
   GP1:
	UF : 0, UT : 1,		CONFIG : 'N U T, 0, 0, 0',
	X = 1218.166  mm,	Y = 121.375  mm,	Z = -237.815  mm,
	W = 0.000 deg,	P = 30.000 deg,	R = 177.800 deg
};
P[370]{
   GP1:
	UF : 0, UT : 1,		CONFIG : 'N U T, 0, 0, 0',
	X = 1224.238  mm,	Y = 123.143  mm,	Z = -237.802  mm,
	W = 0.000 deg,	P = 30.000 deg,	R = 177.800 deg
};
P[371]{
   GP1:
	UF : 0, UT : 1,		CONFIG : 'N U T, 0, 0, 0',
	X = 1224.315  mm,	Y = 125.141  mm,	Z = -237.789  mm,
	W = 0.000 deg,	P = 30.000 deg,	R = 177.800 deg
};
P[372]{
   GP1:
	UF : 0, UT : 1,		CONFIG : 'N U T, 0, 0, 0',
	X = 1224.392  mm,	Y = 127.140  mm,	Z = -237.775  mm,
	W = 0.000 deg,	P = 30.000 deg,	R = 177.800 deg
};
P[373]{
   GP1:
	UF : 0, UT : 1,		CONFIG : 'N U T, 0, 0, 0',
	X = 1224.469  mm,	Y = 129.138  mm,	Z = -237.762  mm,
	W = 0.000 deg,	P = 30.000 deg,	R = 177.800 deg
};
P[374]{
   GP1:
	UF : 0, UT : 1,		CONFIG : 'N U T, 0, 0, 0',
	X = 1224.546  mm,	Y = 131.137  mm,	Z = -237.749  mm,
	W = 0.000 deg,	P = 30.000 deg,	R = 177.800 deg
};
P[375]{
   GP1:
	UF : 0, UT : 1,		CONFIG : 'N U T, 0, 0, 0',
	X = 1224.622  mm,	Y = 133.135  mm,	Z = -237.735  mm,
	W = 0.000 deg,	P = 30.000 deg,	R = 177.800 deg
};
P[376]{
   GP1:
	UF : 0, UT : 1,		CONFIG : 'N U T, 0, 0, 0',
	X = 1224.699  mm,	Y = 135.134  mm,	Z = -237.722  mm,
	W = 0.000 deg,	P = 30.000 deg,	R = 177.800 deg
};
P[377]{
   GP1:
	UF : 0, UT : 1,		CONFIG : 'N U T, 0, 0, 0',
	X = 1224.776  mm,	Y = 137.132  mm,	Z = -237.709  mm,
	W = 0.000 deg,	P = 30.000 deg,	R = 177.800 deg
};
P[378]{
   GP1:
	UF : 0, UT : 1,		CONFIG : 'N U T, 0, 0, 0',
	X = 1224.853  mm,	Y = 139.131  mm,	Z = -237.695  mm,
	W = 0.000 deg,	P = 30.000 deg,	R = 177.800 deg
};
P[379]{
   GP1:
	UF : 0, UT : 1,		CONFIG : 'N U T, 0, 0, 0',
	X = 1224.929  mm,	Y = 141.129  mm,	Z = -237.682  mm,
	W = 0.000 deg,	P = 30.000 deg,	R = 177.800 deg
};
P[380]{
   GP1:
	UF : 0, UT : 1,		CONFIG : 'N U T, 0, 0, 0',
	X = 1225.006  mm,	Y = 143.128  mm,	Z = -237.669  mm,
	W = 0.000 deg,	P = 30.000 deg,	R = 177.800 deg
};
P[381]{
   GP1:
	UF : 0, UT : 1,		CONFIG : 'N U T, 0, 0, 0',
	X = 1225.083  mm,	Y = 145.126  mm,	Z = -237.656  mm,
	W = 0.000 deg,	P = 30.000 deg,	R = 177.800 deg
};
P[382]{
   GP1:
	UF : 0, UT : 1,		CONFIG : 'N U T, 0, 0, 0',
	X = 1219.164  mm,	Y = 147.355  mm,	Z = -237.642  mm,
	W = 0.000 deg,	P = 30.000 deg,	R = 177.800 deg
};
P[383]{
   GP1:
	UF : 0, UT : 1,		CONFIG : 'N U T, 0, 0, 0',
	X = 1225.237  mm,	Y = 149.123  mm,	Z = -237.629  mm,
	W = 0.000 deg,	P = 30.000 deg,	R = 177.800 deg
};
P[384]{
   GP1:
	UF : 0, UT : 1,		CONFIG : 'N U T, 0, 0, 0',
	X = 1219.318  mm,	Y = 151.352  mm,	Z = -237.616  mm,
	W = 0.000 deg,	P = 30.000 deg,	R = 167.603 deg
};
P[385]{
   GP1:
	UF : 0, UT : 1,		CONFIG : 'N U T, 0, 0, 0',
	X = 1219.394  mm,	Y = 153.350  mm,	Z = -237.602  mm,
	W = 0.000 deg,	P = 30.000 deg,	R = 159.869 deg
};
P[386]{
   GP1:
	UF : 0, UT : 1,		CONFIG : 'N U T, 0, 0, 0',
	X = 1219.471  mm,	Y = 155.349  mm,	Z = -237.589  mm,
	W = 0.000 deg,	P = 30.000 deg,	R = 152.135 deg
};
P[387]{
   GP1:
	UF : 0, UT : 1,		CONFIG : 'N U T, 0, 0, 0',
	X = 1219.548  mm,	Y = 157.347  mm,	Z = -237.576  mm,
	W = 0.000 deg,	P = 30.000 deg,	R = 144.400 deg
};
P[388]{
   GP1:
	UF : 0, UT : 1,		CONFIG : 'N U T, 0, 0, 0',
	X = 1219.660  mm,	Y = 159.330  mm,	Z = -237.566  mm,
	W = 0.000 deg,	P = 30.000 deg,	R = 139.128 deg
};
P[389]{
   GP1:
	UF : 0, UT : 1,		CONFIG : 'N U T, 0, 0, 0',
	X = 1220.643  mm,	Y = 161.076  mm,	Z = -237.628  mm,
	W = 0.000 deg,	P = 30.000 deg,	R = 139.128 deg
};
P[390]{
   GP1:
	UF : 0, UT : 1,		CONFIG : 'N U T, 0, 0, 0',
	X = 1221.941  mm,	Y = 162.575  mm,	Z = -237.889  mm,
	W = 0.000 deg,	P = 30.000 deg,	R = 139.128 deg
};
P[391]{
   GP1:
	UF : 0, UT : 1,		CONFIG : 'N U T, 0, 0, 0',
	X = 1223.238  mm,	Y = 164.074  mm,	Z = -238.151  mm,
	W = 0.000 deg,	P = 30.000 deg,	R = 139.128 deg
};
P[392]{
   GP1:
	UF : 0, UT : 1,		CONFIG : 'N U T, 0, 0, 0',
	X = 1229.073  mm,	Y = 161.647  mm,	Z = -238.413  mm,
	W = 0.000 deg,	P = 30.000 deg,	R = 139.128 deg
};
P[393]{
   GP1:
	UF : 0, UT : 1,		CONFIG : 'N U T, 0, 0, 0',
	X = 1230.370  mm,	Y = 163.147  mm,	Z = -238.674  mm,
	W = 0.000 deg,	P = 30.000 deg,	R = 139.128 deg
};
P[394]{
   GP1:
	UF : 0, UT : 1,		CONFIG : 'N U T, 0, 0, 0',
	X = 1227.130  mm,	Y = 168.572  mm,	Z = -238.936  mm,
	W = 0.000 deg,	P = 30.000 deg,	R = 139.128 deg
};
P[395]{
   GP1:
	UF : 0, UT : 1,		CONFIG : 'N U T, 0, 0, 0',
	X = 1232.965  mm,	Y = 166.145  mm,	Z = -239.198  mm,
	W = 0.000 deg,	P = 30.000 deg,	R = 139.128 deg
};
P[396]{
   GP1:
	UF : 0, UT : 1,		CONFIG : 'N U T, 0, 0, 0',
	X = 1234.263  mm,	Y = 167.645  mm,	Z = -239.459  mm,
	W = 0.000 deg,	P = 30.000 deg,	R = 139.128 deg
};
P[397]{
   GP1:
	UF : 0, UT : 1,		CONFIG : 'N U T, 0, 0, 0',
	X = 1235.560  mm,	Y = 169.144  mm,	Z = -239.721  mm,
	W = 0.000 deg,	P = 30.000 deg,	R = 139.128 deg
};
P[398]{
   GP1:
	UF : 0, UT : 1,		CONFIG : 'N U T, 0, 0, 0',
	X = 1236.857  mm,	Y = 170.643  mm,	Z = -239.983  mm,
	W = 0.000 deg,	P = 30.000 deg,	R = 139.128 deg
};
P[399]{
   GP1:
	UF : 0, UT : 1,		CONFIG : 'N U T, 0, 0, 0',
	X = 1233.618  mm,	Y = 176.069  mm,	Z = -240.245  mm,
	W = 0.000 deg,	P = 30.000 deg,	R = 139.128 deg
};
P[400]{
   GP1:
	UF : 0, UT : 1,		CONFIG : 'N U T, 0, 0, 0',
	X = 1234.915  mm,	Y = 177.568  mm,	Z = -240.506  mm,
	W = 0.000 deg,	P = 30.000 deg,	R = 139.128 deg
};
P[401]{
   GP1:
	UF : 0, UT : 1,		CONFIG : 'N U T, 0, 0, 0',
	X = 1236.213  mm,	Y = 179.068  mm,	Z = -240.768  mm,
	W = 0.000 deg,	P = 30.000 deg,	R = 139.128 deg
};
P[402]{
   GP1:
	UF : 0, UT : 1,		CONFIG : 'N U T, 0, 0, 0',
	X = 1237.510  mm,	Y = 180.567  mm,	Z = -241.030  mm,
	W = 0.000 deg,	P = 30.000 deg,	R = 139.128 deg
};
P[403]{
   GP1:
	UF : 0, UT : 1,		CONFIG : 'N U T, 0, 0, 0',
	X = 1243.345  mm,	Y = 178.140  mm,	Z = -241.291  mm,
	W = 0.000 deg,	P = 30.000 deg,	R = 139.128 deg
};
P[404]{
   GP1:
	UF : 0, UT : 1,		CONFIG : 'N U T, 0, 0, 0',
	X = 1244.642  mm,	Y = 179.639  mm,	Z = -241.553  mm,
	W = 0.000 deg,	P = 30.000 deg,	R = 139.128 deg
};
P[405]{
   GP1:
	UF : 0, UT : 1,		CONFIG : 'N U T, 0, 0, 0',
	X = 1241.403  mm,	Y = 185.065  mm,	Z = -241.815  mm,
	W = 0.000 deg,	P = 30.000 deg,	R = 139.128 deg
};
P[406]{
   GP1:
	UF : 0, UT : 1,		CONFIG : 'N U T, 0, 0, 0',
	X = 1247.237  mm,	Y = 182.638  mm,	Z = -242.076  mm,
	W = 0.000 deg,	P = 30.000 deg,	R = 139.128 deg
};
P[407]{
   GP1:
	UF : 0, UT : 1,		CONFIG : 'N U T, 0, 0, 0',
	X = 1248.535  mm,	Y = 184.138  mm,	Z = -242.338  mm,
	W = 0.000 deg,	P = 30.000 deg,	R = 139.128 deg
};
P[408]{
   GP1:
	UF : 0, UT : 1,		CONFIG : 'N U T, 0, 0, 0',
	X = 1249.832  mm,	Y = 185.637  mm,	Z = -242.600  mm,
	W = 0.000 deg,	P = 30.000 deg,	R = 139.128 deg
};
P[409]{
   GP1:
	UF : 0, UT : 1,		CONFIG : 'N U T, 0, 0, 0',
	X = 1251.130  mm,	Y = 187.136  mm,	Z = -242.862  mm,
	W = 0.000 deg,	P = 30.000 deg,	R = 139.128 deg
};
P[410]{
   GP1:
	UF : 0, UT : 1,		CONFIG : 'N U T, 0, 0, 0',
	X = 1247.890  mm,	Y = 192.562  mm,	Z = -243.123  mm,
	W = 0.000 deg,	P = 30.000 deg,	R = 139.128 deg
};
P[411]{
   GP1:
	UF : 0, UT : 1,		CONFIG : 'N U T, 0, 0, 0',
	X = 1249.188  mm,	Y = 194.061  mm,	Z = -243.385  mm,
	W = 0.000 deg,	P = 30.000 deg,	R = 139.128 deg
};
P[412]{
   GP1:
	UF : 0, UT : 1,		CONFIG : 'N U T, 0, 0, 0',
	X = 1255.022  mm,	Y = 191.634  mm,	Z = -243.647  mm,
	W = 0.000 deg,	P = 30.000 deg,	R = 148.871 deg
};
P[413]{
   GP1:
	UF : 0, UT : 1,		CONFIG : 'N U T, 0, 0, 0',
	X = 1256.320  mm,	Y = 193.134  mm,	Z = -243.908  mm,
	W = 0.000 deg,	P = 30.000 deg,	R = 156.748 deg
};
P[414]{
   GP1:
	UF : 0, UT : 1,		CONFIG : 'N U T, 0, 0, 0',
	X = 1257.617  mm,	Y = 194.633  mm,	Z = -244.170  mm,
	W = 0.000 deg,	P = 30.000 deg,	R = 164.626 deg
};
P[415]{
   GP1:
	UF : 0, UT : 1,		CONFIG : 'N U T, 0, 0, 0',
	X = 1258.915  mm,	Y = 196.132  mm,	Z = -244.432  mm,
	W = 0.000 deg,	P = 30.000 deg,	R = 172.503 deg
};
P[416]{
   GP1:
	UF : 0, UT : 1,		CONFIG : 'N U T, 0, 0, 0',
	X = 1260.212  mm,	Y = 197.632  mm,	Z = -244.693  mm,
	W = 0.000 deg,	P = 30.000 deg,	R = 178.516 deg
};
P[417]{
   GP1:
	UF : 0, UT : 1,		CONFIG : 'N U T, 0, 0, 0',
	X = 1261.427  mm,	Y = 199.228  mm,	Z = -244.844  mm,
	W = 0.000 deg,	P = 30.000 deg,	R = 178.516 deg
};
P[418]{
   GP1:
	UF : 0, UT : 1,		CONFIG : 'N U T, 0, 0, 0',
	X = 1255.714  mm,	Y = 201.384  mm,	Z = -244.837  mm,
	W = 0.000 deg,	P = 30.000 deg,	R = 178.516 deg
};
P[419]{
   GP1:
	UF : 0, UT : 1,		CONFIG : 'N U T, 0, 0, 0',
	X = 1255.766  mm,	Y = 203.383  mm,	Z = -244.819  mm,
	W = 0.000 deg,	P = 30.000 deg,	R = 178.516 deg
};
P[420]{
   GP1:
	UF : 0, UT : 1,		CONFIG : 'N U T, 0, 0, 0',
	X = 1261.815  mm,	Y = 205.227  mm,	Z = -244.801  mm,
	W = 0.000 deg,	P = 30.000 deg,	R = 178.516 deg
};
P[421]{
   GP1:
	UF : 0, UT : 1,		CONFIG : 'N U T, 0, 0, 0',
	X = 1255.869  mm,	Y = 207.382  mm,	Z = -244.783  mm,
	W = 0.000 deg,	P = 30.000 deg,	R = 178.516 deg
};
P[422]{
   GP1:
	UF : 0, UT : 1,		CONFIG : 'N U T, 0, 0, 0',
	X = 1255.921  mm,	Y = 209.381  mm,	Z = -244.765  mm,
	W = 0.000 deg,	P = 30.000 deg,	R = 178.516 deg
};
P[423]{
   GP1:
	UF : 0, UT : 1,		CONFIG : 'N U T, 0, 0, 0',
	X = 1255.973  mm,	Y = 211.380  mm,	Z = -244.747  mm,
	W = 0.000 deg,	P = 30.000 deg,	R = 178.516 deg
};
P[424]{
   GP1:
	UF : 0, UT : 1,		CONFIG : 'N U T, 0, 0, 0',
	X = 1256.025  mm,	Y = 213.379  mm,	Z = -244.730  mm,
	W = 0.000 deg,	P = 30.000 deg,	R = 178.516 deg
};
P[425]{
   GP1:
	UF : 0, UT : 1,		CONFIG : 'N U T, 0, 0, 0',
	X = 1256.076  mm,	Y = 215.379  mm,	Z = -244.712  mm,
	W = 0.000 deg,	P = 30.000 deg,	R = 178.516 deg
};
P[426]{
   GP1:
	UF : 0, UT : 1,		CONFIG : 'N U T, 0, 0, 0',
	X = 1256.128  mm,	Y = 217.378  mm,	Z = -244.694  mm,
	W = 0.000 deg,	P = 30.000 deg,	R = 178.516 deg
};
P[427]{
   GP1:
	UF : 0, UT : 1,		CONFIG : 'N U T, 0, 0, 0',
	X = 1256.180  mm,	Y = 219.377  mm,	Z = -244.676  mm,
	W = 0.000 deg,	P = 30.000 deg,	R = 178.516 deg
};
P[428]{
   GP1:
	UF : 0, UT : 1,		CONFIG : 'N U T, 0, 0, 0',
	X = 1262.230  mm,	Y = 221.221  mm,	Z = -244.658  mm,
	W = 0.000 deg,	P = 30.000 deg,	R = 178.516 deg
};
P[429]{
   GP1:
	UF : 0, UT : 1,		CONFIG : 'N U T, 0, 0, 0',
	X = 1262.260  mm,	Y = 222.372  mm,	Z = -244.648  mm,
	W = 0.000 deg,	P = 30.000 deg,	R = 178.516 deg
};
/END
